;ENDFOLD
;FOLD LIN P193 CONT Vel=1 m/s CPDATP193 Tool[2] Base[10] ;%{PE}
;FOLD Parameters ;%{h}
;Params IlfProvider=kukaroboter.basistech.inlineforms.movement.old; Kuka.IsGlobalPoint=False; Kuka.PointName=P193; Kuka.BlendingEnabled=TRUE; Kuka.MoveDataName=CPDATP193; Kuka.VelocityPath=1; Kuka.CurrentCDSetIndex=0; Kuka.MovementParameterFieldEnabled=True; IlfCommand=LIN
;ENDFOLD
$BWDSTART = FALSE
LDAT_ACT=LCPDATP193
FDAT_ACT=FP193
BAS (#CP_PARAMS,1)
SET_CD_PARAMS (0)
LIN XP193 C_DIS

;ENDFOLD
;FOLD CIRC CAux194 CDes194 CONT Vel=0.1 m/s CPDATC194 Tool[2] Base[10] ;%{PE}
;FOLD Parameters ;%{h}
;Params IlfProvider=kukaroboter.basistech.inlineforms.movement.old; Kuka.IsGlobalPoint=False; Kuka.PointName=CDes194; Kuka.BlendingEnabled=TRUE; Kuka.MoveDataName=CPDATC194; Kuka.VelocityPath=0.1; Kuka.CurrentCDSetIndex=0; Kuka.MovementParameterFieldEnabled=True; IlfCommand=LIN
;ENDFOLD
$BWDSTART = FALSE
LDAT_ACT=LCPDATC194
FDAT_ACT=FC194
$ORI_TYPE = #VAR
$CIRC_TYPE = #PATH
BAS (#CP_PARAMS,0.1)
SET_CD_PARAMS (0)
CIRC XCAux194, XCDes194 C_DIS

;ENDFOLD
;FOLD LIN P195 CONT Vel=1 m/s CPDATP195 Tool[2] Base[10] ;%{PE}
;FOLD Parameters ;%{h}
;Params IlfProvider=kukaroboter.basistech.inlineforms.movement.old; Kuka.IsGlobalPoint=False; Kuka.PointName=P195; Kuka.BlendingEnabled=TRUE; Kuka.MoveDataName=CPDATP195; Kuka.VelocityPath=1; Kuka.CurrentCDSetIndex=0; Kuka.MovementParameterFieldEnabled=True; IlfCommand=LIN
;ENDFOLD
$BWDSTART = FALSE
LDAT_ACT=LCPDATP195
FDAT_ACT=FP195
BAS (#CP_PARAMS,1)
SET_CD_PARAMS (0)
LIN XP195 C_DIS

;ENDFOLD
;FOLD LIN P196 CONT Vel=1 m/s CPDATP196 Tool[2] Base[10] ;%{PE}
;FOLD Parameters ;%{h}
;Params IlfProvider=kukaroboter.basistech.inlineforms.movement.old; Kuka.IsGlobalPoint=False; Kuka.PointName=P196; Kuka.BlendingEnabled=TRUE; Kuka.MoveDataName=CPDATP196; Kuka.VelocityPath=1; Kuka.CurrentCDSetIndex=0; Kuka.MovementParameterFieldEnabled=True; IlfCommand=LIN
;ENDFOLD
$BWDSTART = FALSE
LDAT_ACT=LCPDATP196
FDAT_ACT=FP196
BAS (#CP_PARAMS,1)
SET_CD_PARAMS (0)
LIN XP196 C_DIS

;ENDFOLD
;FOLD CIRC CAux197 CDes197 CONT Vel=0.1 m/s CPDATC197 Tool[2] Base[10] ;%{PE}
;FOLD Parameters ;%{h}
;Params IlfProvider=kukaroboter.basistech.inlineforms.movement.old; Kuka.IsGlobalPoint=False; Kuka.PointName=CDes197; Kuka.BlendingEnabled=TRUE; Kuka.MoveDataName=CPDATC197; Kuka.VelocityPath=0.1; Kuka.CurrentCDSetIndex=0; Kuka.MovementParameterFieldEnabled=True; IlfCommand=LIN
;ENDFOLD
$BWDSTART = FALSE
LDAT_ACT=LCPDATC197
FDAT_ACT=FC197
$ORI_TYPE = #VAR
$CIRC_TYPE = #PATH
BAS (#CP_PARAMS,0.1)
SET_CD_PARAMS (0)
CIRC XCAux197, XCDes197 C_DIS

;ENDFOLD
;FOLD LIN P198 CONT Vel=1 m/s CPDATP198 Tool[2] Base[10] ;%{PE}
;FOLD Parameters ;%{h}
;Params IlfProvider=kukaroboter.basistech.inlineforms.movement.old; Kuka.IsGlobalPoint=False; Kuka.PointName=P198; Kuka.BlendingEnabled=TRUE; Kuka.MoveDataName=CPDATP198; Kuka.VelocityPath=1; Kuka.CurrentCDSetIndex=0; Kuka.MovementParameterFieldEnabled=True; IlfCommand=LIN
;ENDFOLD
$BWDSTART = FALSE
LDAT_ACT=LCPDATP198
FDAT_ACT=FP198
BAS (#CP_PARAMS,1)
SET_CD_PARAMS (0)
LIN XP198 C_DIS

;ENDFOLD
;FOLD LIN P199 CONT Vel=1 m/s CPDATP199 Tool[2] Base[10] ;%{PE}
;FOLD Parameters ;%{h}
;Params IlfProvider=kukaroboter.basistech.inlineforms.movement.old; Kuka.IsGlobalPoint=False; Kuka.PointName=P199; Kuka.BlendingEnabled=TRUE; Kuka.MoveDataName=CPDATP199; Kuka.VelocityPath=1; Kuka.CurrentCDSetIndex=0; Kuka.MovementParameterFieldEnabled=True; IlfCommand=LIN
;ENDFOLD
$BWDSTART = FALSE
LDAT_ACT=LCPDATP199
FDAT_ACT=FP199
BAS (#CP_PARAMS,1)
SET_CD_PARAMS (0)
LIN XP199 C_DIS

;ENDFOLD
;FOLD CIRC CAux200 CDes200 CONT Vel=0.1 m/s CPDATC200 Tool[2] Base[10] ;%{PE}
;FOLD Parameters ;%{h}
;Params IlfProvider=kukaroboter.basistech.inlineforms.movement.old; Kuka.IsGlobalPoint=False; Kuka.PointName=CDes200; Kuka.BlendingEnabled=TRUE; Kuka.MoveDataName=CPDATC200; Kuka.VelocityPath=0.1; Kuka.CurrentCDSetIndex=0; Kuka.MovementParameterFieldEnabled=True; IlfCommand=LIN
;ENDFOLD
$BWDSTART = FALSE
LDAT_ACT=LCPDATC200
FDAT_ACT=FC200
$ORI_TYPE = #VAR
$CIRC_TYPE = #PATH
BAS (#CP_PARAMS,0.1)
SET_CD_PARAMS (0)
CIRC XCAux200, XCDes200 C_DIS

;ENDFOLD
;FOLD LIN P201 CONT Vel=1 m/s CPDATP201 Tool[2] Base[10] ;%{PE}
;FOLD Parameters ;%{h}
;Params IlfProvider=kukaroboter.basistech.inlineforms.movement.old; Kuka.IsGlobalPoint=False; Kuka.PointName=P201; Kuka.BlendingEnabled=TRUE; Kuka.MoveDataName=CPDATP201; Kuka.VelocityPath=1; Kuka.CurrentCDSetIndex=0; Kuka.MovementParameterFieldEnabled=True; IlfCommand=LIN
;ENDFOLD
$BWDSTART = FALSE
LDAT_ACT=LCPDATP201
FDAT_ACT=FP201
BAS (#CP_PARAMS,1)
SET_CD_PARAMS (0)
LIN XP201 C_DIS

;ENDFOLD
;FOLD LIN P202 CONT Vel=1 m/s CPDATP202 Tool[2] Base[10] ;%{PE}
;FOLD Parameters ;%{h}
;Params IlfProvider=kukaroboter.basistech.inlineforms.movement.old; Kuka.IsGlobalPoint=False; Kuka.PointName=P202; Kuka.BlendingEnabled=TRUE; Kuka.MoveDataName=CPDATP202; Kuka.VelocityPath=1; Kuka.CurrentCDSetIndex=0; Kuka.MovementParameterFieldEnabled=True; IlfCommand=LIN
;ENDFOLD
$BWDSTART = FALSE
LDAT_ACT=LCPDATP202
FDAT_ACT=FP202
BAS (#CP_PARAMS,1)
SET_CD_PARAMS (0)
LIN XP202 C_DIS

;ENDFOLD
;FOLD CIRC CAux203 CDes203 CONT Vel=0.1 m/s CPDATC203 Tool[2] Base[10] ;%{PE}
;FOLD Parameters ;%{h}
;Params IlfProvider=kukaroboter.basistech.inlineforms.movement.old; Kuka.IsGlobalPoint=False; Kuka.PointName=CDes203; Kuka.BlendingEnabled=TRUE; Kuka.MoveDataName=CPDATC203; Kuka.VelocityPath=0.1; Kuka.CurrentCDSetIndex=0; Kuka.MovementParameterFieldEnabled=True; IlfCommand=LIN
;ENDFOLD
$BWDSTART = FALSE
LDAT_ACT=LCPDATC203
FDAT_ACT=FC203
$ORI_TYPE = #VAR
$CIRC_TYPE = #PATH
BAS (#CP_PARAMS,0.1)
SET_CD_PARAMS (0)
CIRC XCAux203, XCDes203 C_DIS

;ENDFOLD
;FOLD LIN P204 CONT Vel=1 m/s CPDATP204 Tool[2] Base[10] ;%{PE}
;FOLD Parameters ;%{h}
;Params IlfProvider=kukaroboter.basistech.inlineforms.movement.old; Kuka.IsGlobalPoint=False; Kuka.PointName=P204; Kuka.BlendingEnabled=TRUE; Kuka.MoveDataName=CPDATP204; Kuka.VelocityPath=1; Kuka.CurrentCDSetIndex=0; Kuka.MovementParameterFieldEnabled=True; IlfCommand=LIN
;ENDFOLD
$BWDSTART = FALSE
LDAT_ACT=LCPDATP204
FDAT_ACT=FP204
BAS (#CP_PARAMS,1)
SET_CD_PARAMS (0)
LIN XP204 C_DIS

;ENDFOLD
;FOLD LIN P205 CONT Vel=1 m/s CPDATP205 Tool[2] Base[10] ;%{PE}
;FOLD Parameters ;%{h}
;Params IlfProvider=kukaroboter.basistech.inlineforms.movement.old; Kuka.IsGlobalPoint=False; Kuka.PointName=P205; Kuka.BlendingEnabled=TRUE; Kuka.MoveDataName=CPDATP205; Kuka.VelocityPath=1; Kuka.CurrentCDSetIndex=0; Kuka.MovementParameterFieldEnabled=True; IlfCommand=LIN
;ENDFOLD
$BWDSTART = FALSE
LDAT_ACT=LCPDATP205
FDAT_ACT=FP205
BAS (#CP_PARAMS,1)
SET_CD_PARAMS (0)
LIN XP205 C_DIS

;ENDFOLD
;FOLD CIRC CAux206 CDes206 CONT Vel=0.1 m/s CPDATC206 Tool[2] Base[10] ;%{PE}
;FOLD Parameters ;%{h}
;Params IlfProvider=kukaroboter.basistech.inlineforms.movement.old; Kuka.IsGlobalPoint=False; Kuka.PointName=CDes206; Kuka.BlendingEnabled=TRUE; Kuka.MoveDataName=CPDATC206; Kuka.VelocityPath=0.1; Kuka.CurrentCDSetIndex=0; Kuka.MovementParameterFieldEnabled=True; IlfCommand=LIN
;ENDFOLD
$BWDSTART = FALSE
LDAT_ACT=LCPDATC206
FDAT_ACT=FC206
$ORI_TYPE = #VAR
$CIRC_TYPE = #PATH
BAS (#CP_PARAMS,0.1)
SET_CD_PARAMS (0)
CIRC XCAux206, XCDes206 C_DIS

;ENDFOLD
;FOLD LIN P207 CONT Vel=1 m/s CPDATP207 Tool[2] Base[10] ;%{PE}
;FOLD Parameters ;%{h}
;Params IlfProvider=kukaroboter.basistech.inlineforms.movement.old; Kuka.IsGlobalPoint=False; Kuka.PointName=P207; Kuka.BlendingEnabled=TRUE; Kuka.MoveDataName=CPDATP207; Kuka.VelocityPath=1; Kuka.CurrentCDSetIndex=0; Kuka.MovementParameterFieldEnabled=True; IlfCommand=LIN
;ENDFOLD
$BWDSTART = FALSE
LDAT_ACT=LCPDATP207
FDAT_ACT=FP207
BAS (#CP_PARAMS,1)
SET_CD_PARAMS (0)
LIN XP207 C_DIS

;ENDFOLD
;FOLD LIN P208 CONT Vel=1 m/s CPDATP208 Tool[2] Base[10] ;%{PE}
;FOLD Parameters ;%{h}
;Params IlfProvider=kukaroboter.basistech.inlineforms.movement.old; Kuka.IsGlobalPoint=False; Kuka.PointName=P208; Kuka.BlendingEnabled=TRUE; Kuka.MoveDataName=CPDATP208; Kuka.VelocityPath=1; Kuka.CurrentCDSetIndex=0; Kuka.MovementParameterFieldEnabled=True; IlfCommand=LIN
;ENDFOLD
$BWDSTART = FALSE
LDAT_ACT=LCPDATP208
FDAT_ACT=FP208
BAS (#CP_PARAMS,1)
SET_CD_PARAMS (0)
LIN XP208 C_DIS

;ENDFOLD
;FOLD CIRC CAux209 CDes209 CONT Vel=0.1 m/s CPDATC209 Tool[2] Base[10] ;%{PE}
;FOLD Parameters ;%{h}
;Params IlfProvider=kukaroboter.basistech.inlineforms.movement.old; Kuka.IsGlobalPoint=False; Kuka.PointName=CDes209; Kuka.BlendingEnabled=TRUE; Kuka.MoveDataName=CPDATC209; Kuka.VelocityPath=0.1; Kuka.CurrentCDSetIndex=0; Kuka.MovementParameterFieldEnabled=True; IlfCommand=LIN
;ENDFOLD
$BWDSTART = FALSE
LDAT_ACT=LCPDATC209
FDAT_ACT=FC209
$ORI_TYPE = #VAR
$CIRC_TYPE = #PATH
BAS (#CP_PARAMS,0.1)
SET_CD_PARAMS (0)
CIRC XCAux209, XCDes209 C_DIS

;ENDFOLD
;FOLD LIN P210 CONT Vel=1 m/s CPDATP210 Tool[2] Base[10] ;%{PE}
;FOLD Parameters ;%{h}
;Params IlfProvider=kukaroboter.basistech.inlineforms.movement.old; Kuka.IsGlobalPoint=False; Kuka.PointName=P210; Kuka.BlendingEnabled=TRUE; Kuka.MoveDataName=CPDATP210; Kuka.VelocityPath=1; Kuka.CurrentCDSetIndex=0; Kuka.MovementParameterFieldEnabled=True; IlfCommand=LIN
;ENDFOLD
$BWDSTART = FALSE
LDAT_ACT=LCPDATP210
FDAT_ACT=FP210
BAS (#CP_PARAMS,1)
SET_CD_PARAMS (0)
LIN XP210 C_DIS

;ENDFOLD
;FOLD LIN P211 CONT Vel=1 m/s CPDATP211 Tool[2] Base[10] ;%{PE}
;FOLD Parameters ;%{h}
;Params IlfProvider=kukaroboter.basistech.inlineforms.movement.old; Kuka.IsGlobalPoint=False; Kuka.PointName=P211; Kuka.BlendingEnabled=TRUE; Kuka.MoveDataName=CPDATP211; Kuka.VelocityPath=1; Kuka.CurrentCDSetIndex=0; Kuka.MovementParameterFieldEnabled=True; IlfCommand=LIN
;ENDFOLD
$BWDSTART = FALSE
LDAT_ACT=LCPDATP211
FDAT_ACT=FP211
BAS (#CP_PARAMS,1)
SET_CD_PARAMS (0)
LIN XP211 C_DIS

;ENDFOLD
;FOLD CIRC CAux212 CDes212 CONT Vel=0.1 m/s CPDATC212 Tool[2] Base[10] ;%{PE}
;FOLD Parameters ;%{h}
;Params IlfProvider=kukaroboter.basistech.inlineforms.movement.old; Kuka.IsGlobalPoint=False; Kuka.PointName=CDes212; Kuka.BlendingEnabled=TRUE; Kuka.MoveDataName=CPDATC212; Kuka.VelocityPath=0.1; Kuka.CurrentCDSetIndex=0; Kuka.MovementParameterFieldEnabled=True; IlfCommand=LIN
;ENDFOLD
$BWDSTART = FALSE
LDAT_ACT=LCPDATC212
FDAT_ACT=FC212
$ORI_TYPE = #VAR
$CIRC_TYPE = #PATH
BAS (#CP_PARAMS,0.1)
SET_CD_PARAMS (0)
CIRC XCAux212, XCDes212 C_DIS

;ENDFOLD
;FOLD LIN P213 CONT Vel=1 m/s CPDATP213 Tool[2] Base[10] ;%{PE}
;FOLD Parameters ;%{h}
;Params IlfProvider=kukaroboter.basistech.inlineforms.movement.old; Kuka.IsGlobalPoint=False; Kuka.PointName=P213; Kuka.BlendingEnabled=TRUE; Kuka.MoveDataName=CPDATP213; Kuka.VelocityPath=1; Kuka.CurrentCDSetIndex=0; Kuka.MovementParameterFieldEnabled=True; IlfCommand=LIN
;ENDFOLD
$BWDSTART = FALSE
LDAT_ACT=LCPDATP213
FDAT_ACT=FP213
BAS (#CP_PARAMS,1)
SET_CD_PARAMS (0)
LIN XP213 C_DIS

;ENDFOLD
;FOLD LIN P214 CONT Vel=1 m/s CPDATP214 Tool[2] Base[10] ;%{PE}
;FOLD Parameters ;%{h}
;Params IlfProvider=kukaroboter.basistech.inlineforms.movement.old; Kuka.IsGlobalPoint=False; Kuka.PointName=P214; Kuka.BlendingEnabled=TRUE; Kuka.MoveDataName=CPDATP214; Kuka.VelocityPath=1; Kuka.CurrentCDSetIndex=0; Kuka.MovementParameterFieldEnabled=True; IlfCommand=LIN
;ENDFOLD
$BWDSTART = FALSE
LDAT_ACT=LCPDATP214
FDAT_ACT=FP214
BAS (#CP_PARAMS,1)
SET_CD_PARAMS (0)
LIN XP214 C_DIS

;ENDFOLD
;FOLD CIRC CAux215 CDes215 CONT Vel=0.1 m/s CPDATC215 Tool[2] Base[10] ;%{PE}
;FOLD Parameters ;%{h}
;Params IlfProvider=kukaroboter.basistech.inlineforms.movement.old; Kuka.IsGlobalPoint=False; Kuka.PointName=CDes215; Kuka.BlendingEnabled=TRUE; Kuka.MoveDataName=CPDATC215; Kuka.VelocityPath=0.1; Kuka.CurrentCDSetIndex=0; Kuka.MovementParameterFieldEnabled=True; IlfCommand=LIN
;ENDFOLD
$BWDSTART = FALSE
LDAT_ACT=LCPDATC215
FDAT_ACT=FC215
$ORI_TYPE = #VAR
$CIRC_TYPE = #PATH
BAS (#CP_PARAMS,0.1)
SET_CD_PARAMS (0)
CIRC XCAux215, XCDes215 C_DIS

;ENDFOLD
;FOLD LIN P216 CONT Vel=1 m/s CPDATP216 Tool[2] Base[10] ;%{PE}
;FOLD Parameters ;%{h}
;Params IlfProvider=kukaroboter.basistech.inlineforms.movement.old; Kuka.IsGlobalPoint=False; Kuka.PointName=P216; Kuka.BlendingEnabled=TRUE; Kuka.MoveDataName=CPDATP216; Kuka.VelocityPath=1; Kuka.CurrentCDSetIndex=0; Kuka.MovementParameterFieldEnabled=True; IlfCommand=LIN
;ENDFOLD
$BWDSTART = FALSE
LDAT_ACT=LCPDATP216
FDAT_ACT=FP216
BAS (#CP_PARAMS,1)
SET_CD_PARAMS (0)
LIN XP216 C_DIS

;ENDFOLD
;FOLD LIN P217 CONT Vel=1 m/s CPDATP217 Tool[2] Base[10] ;%{PE}
;FOLD Parameters ;%{h}
;Params IlfProvider=kukaroboter.basistech.inlineforms.movement.old; Kuka.IsGlobalPoint=False; Kuka.PointName=P217; Kuka.BlendingEnabled=TRUE; Kuka.MoveDataName=CPDATP217; Kuka.VelocityPath=1; Kuka.CurrentCDSetIndex=0; Kuka.MovementParameterFieldEnabled=True; IlfCommand=LIN
;ENDFOLD
$BWDSTART = FALSE
LDAT_ACT=LCPDATP217
FDAT_ACT=FP217
BAS (#CP_PARAMS,1)
SET_CD_PARAMS (0)
LIN XP217 C_DIS

;ENDFOLD
;FOLD CIRC CAux218 CDes218 CONT Vel=0.1 m/s CPDATC218 Tool[2] Base[10] ;%{PE}
;FOLD Parameters ;%{h}
;Params IlfProvider=kukaroboter.basistech.inlineforms.movement.old; Kuka.IsGlobalPoint=False; Kuka.PointName=CDes218; Kuka.BlendingEnabled=TRUE; Kuka.MoveDataName=CPDATC218; Kuka.VelocityPath=0.1; Kuka.CurrentCDSetIndex=0; Kuka.MovementParameterFieldEnabled=True; IlfCommand=LIN
;ENDFOLD
$BWDSTART = FALSE
LDAT_ACT=LCPDATC218
FDAT_ACT=FC218
$ORI_TYPE = #VAR
$CIRC_TYPE = #PATH
BAS (#CP_PARAMS,0.1)
SET_CD_PARAMS (0)
CIRC XCAux218, XCDes218 C_DIS

;ENDFOLD
;FOLD LIN P219 CONT Vel=1 m/s CPDATP219 Tool[2] Base[10] ;%{PE}
;FOLD Parameters ;%{h}
;Params IlfProvider=kukaroboter.basistech.inlineforms.movement.old; Kuka.IsGlobalPoint=False; Kuka.PointName=P219; Kuka.BlendingEnabled=TRUE; Kuka.MoveDataName=CPDATP219; Kuka.VelocityPath=1; Kuka.CurrentCDSetIndex=0; Kuka.MovementParameterFieldEnabled=True; IlfCommand=LIN
;ENDFOLD
$BWDSTART = FALSE
LDAT_ACT=LCPDATP219
FDAT_ACT=FP219
BAS (#CP_PARAMS,1)
SET_CD_PARAMS (0)
LIN XP219 C_DIS

;ENDFOLD
;FOLD LIN P220 CONT Vel=1 m/s CPDATP220 Tool[2] Base[10] ;%{PE}
;FOLD Parameters ;%{h}
;Params IlfProvider=kukaroboter.basistech.inlineforms.movement.old; Kuka.IsGlobalPoint=False; Kuka.PointName=P220; Kuka.BlendingEnabled=TRUE; Kuka.MoveDataName=CPDATP220; Kuka.VelocityPath=1; Kuka.CurrentCDSetIndex=0; Kuka.MovementParameterFieldEnabled=True; IlfCommand=LIN
;ENDFOLD
$BWDSTART = FALSE
LDAT_ACT=LCPDATP220
FDAT_ACT=FP220
BAS (#CP_PARAMS,1)
SET_CD_PARAMS (0)
LIN XP220 C_DIS

;ENDFOLD
;FOLD CIRC CAux221 CDes221 CONT Vel=0.1 m/s CPDATC221 Tool[2] Base[10] ;%{PE}
;FOLD Parameters ;%{h}
;Params IlfProvider=kukaroboter.basistech.inlineforms.movement.old; Kuka.IsGlobalPoint=False; Kuka.PointName=CDes221; Kuka.BlendingEnabled=TRUE; Kuka.MoveDataName=CPDATC221; Kuka.VelocityPath=0.1; Kuka.CurrentCDSetIndex=0; Kuka.MovementParameterFieldEnabled=True; IlfCommand=LIN
;ENDFOLD
$BWDSTART = FALSE
LDAT_ACT=LCPDATC221
FDAT_ACT=FC221
$ORI_TYPE = #VAR
$CIRC_TYPE = #PATH
BAS (#CP_PARAMS,0.1)
SET_CD_PARAMS (0)
CIRC XCAux221, XCDes221 C_DIS

;ENDFOLD
;FOLD LIN P222 CONT Vel=1 m/s CPDATP222 Tool[2] Base[10] ;%{PE}
;FOLD Parameters ;%{h}
;Params IlfProvider=kukaroboter.basistech.inlineforms.movement.old; Kuka.IsGlobalPoint=False; Kuka.PointName=P222; Kuka.BlendingEnabled=TRUE; Kuka.MoveDataName=CPDATP222; Kuka.VelocityPath=1; Kuka.CurrentCDSetIndex=0; Kuka.MovementParameterFieldEnabled=True; IlfCommand=LIN
;ENDFOLD
$BWDSTART = FALSE
LDAT_ACT=LCPDATP222
FDAT_ACT=FP222
BAS (#CP_PARAMS,1)
SET_CD_PARAMS (0)
LIN XP222 C_DIS

;ENDFOLD
;FOLD LIN P223 CONT Vel=1 m/s CPDATP223 Tool[2] Base[10] ;%{PE}
;FOLD Parameters ;%{h}
;Params IlfProvider=kukaroboter.basistech.inlineforms.movement.old; Kuka.IsGlobalPoint=False; Kuka.PointName=P223; Kuka.BlendingEnabled=TRUE; Kuka.MoveDataName=CPDATP223; Kuka.VelocityPath=1; Kuka.CurrentCDSetIndex=0; Kuka.MovementParameterFieldEnabled=True; IlfCommand=LIN
;ENDFOLD
$BWDSTART = FALSE
LDAT_ACT=LCPDATP223
FDAT_ACT=FP223
BAS (#CP_PARAMS,1)
SET_CD_PARAMS (0)
LIN XP223 C_DIS

;ENDFOLD
;FOLD CIRC CAux224 CDes224 CONT Vel=0.1 m/s CPDATC224 Tool[2] Base[10] ;%{PE}
;FOLD Parameters ;%{h}
;Params IlfProvider=kukaroboter.basistech.inlineforms.movement.old; Kuka.IsGlobalPoint=False; Kuka.PointName=CDes224; Kuka.BlendingEnabled=TRUE; Kuka.MoveDataName=CPDATC224; Kuka.VelocityPath=0.1; Kuka.CurrentCDSetIndex=0; Kuka.MovementParameterFieldEnabled=True; IlfCommand=LIN
;ENDFOLD
$BWDSTART = FALSE
LDAT_ACT=LCPDATC224
FDAT_ACT=FC224
$ORI_TYPE = #VAR
$CIRC_TYPE = #PATH
BAS (#CP_PARAMS,0.1)
SET_CD_PARAMS (0)
CIRC XCAux224, XCDes224 C_DIS

;ENDFOLD
;FOLD LIN P225 CONT Vel=1 m/s CPDATP225 Tool[2] Base[10] ;%{PE}
;FOLD Parameters ;%{h}
;Params IlfProvider=kukaroboter.basistech.inlineforms.movement.old; Kuka.IsGlobalPoint=False; Kuka.PointName=P225; Kuka.BlendingEnabled=TRUE; Kuka.MoveDataName=CPDATP225; Kuka.VelocityPath=1; Kuka.CurrentCDSetIndex=0; Kuka.MovementParameterFieldEnabled=True; IlfCommand=LIN
;ENDFOLD
$BWDSTART = FALSE
LDAT_ACT=LCPDATP225
FDAT_ACT=FP225
BAS (#CP_PARAMS,1)
SET_CD_PARAMS (0)
LIN XP225 C_DIS

;ENDFOLD
;FOLD LIN P226 CONT Vel=1 m/s CPDATP226 Tool[2] Base[10] ;%{PE}
;FOLD Parameters ;%{h}
;Params IlfProvider=kukaroboter.basistech.inlineforms.movement.old; Kuka.IsGlobalPoint=False; Kuka.PointName=P226; Kuka.BlendingEnabled=TRUE; Kuka.MoveDataName=CPDATP226; Kuka.VelocityPath=1; Kuka.CurrentCDSetIndex=0; Kuka.MovementParameterFieldEnabled=True; IlfCommand=LIN
;ENDFOLD
$BWDSTART = FALSE
LDAT_ACT=LCPDATP226
FDAT_ACT=FP226
BAS (#CP_PARAMS,1)
SET_CD_PARAMS (0)
LIN XP226 C_DIS

;ENDFOLD
;FOLD CIRC CAux227 CDes227 CONT Vel=0.1 m/s CPDATC227 Tool[2] Base[10] ;%{PE}
;FOLD Parameters ;%{h}
;Params IlfProvider=kukaroboter.basistech.inlineforms.movement.old; Kuka.IsGlobalPoint=False; Kuka.PointName=CDes227; Kuka.BlendingEnabled=TRUE; Kuka.MoveDataName=CPDATC227; Kuka.VelocityPath=0.1; Kuka.CurrentCDSetIndex=0; Kuka.MovementParameterFieldEnabled=True; IlfCommand=LIN
;ENDFOLD
$BWDSTART = FALSE
LDAT_ACT=LCPDATC227
FDAT_ACT=FC227
$ORI_TYPE = #VAR
$CIRC_TYPE = #PATH
BAS (#CP_PARAMS,0.1)
SET_CD_PARAMS (0)
CIRC XCAux227, XCDes227 C_DIS

;ENDFOLD
;FOLD LIN P228 CONT Vel=1 m/s CPDATP228 Tool[2] Base[10] ;%{PE}
;FOLD Parameters ;%{h}
;Params IlfProvider=kukaroboter.basistech.inlineforms.movement.old; Kuka.IsGlobalPoint=False; Kuka.PointName=P228; Kuka.BlendingEnabled=TRUE; Kuka.MoveDataName=CPDATP228; Kuka.VelocityPath=1; Kuka.CurrentCDSetIndex=0; Kuka.MovementParameterFieldEnabled=True; IlfCommand=LIN
;ENDFOLD
$BWDSTART = FALSE
LDAT_ACT=LCPDATP228
FDAT_ACT=FP228
BAS (#CP_PARAMS,1)
SET_CD_PARAMS (0)
LIN XP228 C_DIS

;ENDFOLD
;FOLD LIN P229 CONT Vel=1 m/s CPDATP229 Tool[2] Base[10] ;%{PE}
;FOLD Parameters ;%{h}
;Params IlfProvider=kukaroboter.basistech.inlineforms.movement.old; Kuka.IsGlobalPoint=False; Kuka.PointName=P229; Kuka.BlendingEnabled=TRUE; Kuka.MoveDataName=CPDATP229; Kuka.VelocityPath=1; Kuka.CurrentCDSetIndex=0; Kuka.MovementParameterFieldEnabled=True; IlfCommand=LIN
;ENDFOLD
$BWDSTART = FALSE
LDAT_ACT=LCPDATP229
FDAT_ACT=FP229
BAS (#CP_PARAMS,1)
SET_CD_PARAMS (0)
LIN XP229 C_DIS

;ENDFOLD
;FOLD CIRC CAux230 CDes230 CONT Vel=0.1 m/s CPDATC230 Tool[2] Base[10] ;%{PE}
;FOLD Parameters ;%{h}
;Params IlfProvider=kukaroboter.basistech.inlineforms.movement.old; Kuka.IsGlobalPoint=False; Kuka.PointName=CDes230; Kuka.BlendingEnabled=TRUE; Kuka.MoveDataName=CPDATC230; Kuka.VelocityPath=0.1; Kuka.CurrentCDSetIndex=0; Kuka.MovementParameterFieldEnabled=True; IlfCommand=LIN
;ENDFOLD
$BWDSTART = FALSE
LDAT_ACT=LCPDATC230
FDAT_ACT=FC230
$ORI_TYPE = #VAR
$CIRC_TYPE = #PATH
BAS (#CP_PARAMS,0.1)
SET_CD_PARAMS (0)
CIRC XCAux230, XCDes230 C_DIS

;ENDFOLD
;FOLD LIN P231 CONT Vel=1 m/s CPDATP231 Tool[2] Base[10] ;%{PE}
;FOLD Parameters ;%{h}
;Params IlfProvider=kukaroboter.basistech.inlineforms.movement.old; Kuka.IsGlobalPoint=False; Kuka.PointName=P231; Kuka.BlendingEnabled=TRUE; Kuka.MoveDataName=CPDATP231; Kuka.VelocityPath=1; Kuka.CurrentCDSetIndex=0; Kuka.MovementParameterFieldEnabled=True; IlfCommand=LIN
;ENDFOLD
$BWDSTART = FALSE
LDAT_ACT=LCPDATP231
FDAT_ACT=FP231
BAS (#CP_PARAMS,1)
SET_CD_PARAMS (0)
LIN XP231 C_DIS

;ENDFOLD
;FOLD LIN P232 CONT Vel=1 m/s CPDATP232 Tool[2] Base[10] ;%{PE}
;FOLD Parameters ;%{h}
;Params IlfProvider=kukaroboter.basistech.inlineforms.movement.old; Kuka.IsGlobalPoint=False; Kuka.PointName=P232; Kuka.BlendingEnabled=TRUE; Kuka.MoveDataName=CPDATP232; Kuka.VelocityPath=1; Kuka.CurrentCDSetIndex=0; Kuka.MovementParameterFieldEnabled=True; IlfCommand=LIN
;ENDFOLD
$BWDSTART = FALSE
LDAT_ACT=LCPDATP232
FDAT_ACT=FP232
BAS (#CP_PARAMS,1)
SET_CD_PARAMS (0)
LIN XP232 C_DIS

;ENDFOLD
;FOLD CIRC CAux233 CDes233 CONT Vel=0.1 m/s CPDATC233 Tool[2] Base[10] ;%{PE}
;FOLD Parameters ;%{h}
;Params IlfProvider=kukaroboter.basistech.inlineforms.movement.old; Kuka.IsGlobalPoint=False; Kuka.PointName=CDes233; Kuka.BlendingEnabled=TRUE; Kuka.MoveDataName=CPDATC233; Kuka.VelocityPath=0.1; Kuka.CurrentCDSetIndex=0; Kuka.MovementParameterFieldEnabled=True; IlfCommand=LIN
;ENDFOLD
$BWDSTART = FALSE
LDAT_ACT=LCPDATC233
FDAT_ACT=FC233
$ORI_TYPE = #VAR
$CIRC_TYPE = #PATH
BAS (#CP_PARAMS,0.1)
SET_CD_PARAMS (0)
CIRC XCAux233, XCDes233 C_DIS

;ENDFOLD
;FOLD LIN P234 CONT Vel=1 m/s CPDATP234 Tool[2] Base[10] ;%{PE}
;FOLD Parameters ;%{h}
;Params IlfProvider=kukaroboter.basistech.inlineforms.movement.old; Kuka.IsGlobalPoint=False; Kuka.PointName=P234; Kuka.BlendingEnabled=TRUE; Kuka.MoveDataName=CPDATP234; Kuka.VelocityPath=1; Kuka.CurrentCDSetIndex=0; Kuka.MovementParameterFieldEnabled=True; IlfCommand=LIN
;ENDFOLD
$BWDSTART = FALSE
LDAT_ACT=LCPDATP234
FDAT_ACT=FP234
BAS (#CP_PARAMS,1)
SET_CD_PARAMS (0)
LIN XP234 C_DIS

;ENDFOLD
;FOLD LIN P235 CONT Vel=1 m/s CPDATP235 Tool[2] Base[10] ;%{PE}
;FOLD Parameters ;%{h}
;Params IlfProvider=kukaroboter.basistech.inlineforms.movement.old; Kuka.IsGlobalPoint=False; Kuka.PointName=P235; Kuka.BlendingEnabled=TRUE; Kuka.MoveDataName=CPDATP235; Kuka.VelocityPath=1; Kuka.CurrentCDSetIndex=0; Kuka.MovementParameterFieldEnabled=True; IlfCommand=LIN
;ENDFOLD
$BWDSTART = FALSE
LDAT_ACT=LCPDATP235
FDAT_ACT=FP235
BAS (#CP_PARAMS,1)
SET_CD_PARAMS (0)
LIN XP235 C_DIS

;ENDFOLD
;FOLD CIRC CAux236 CDes236 CONT Vel=0.1 m/s CPDATC236 Tool[2] Base[10] ;%{PE}
;FOLD Parameters ;%{h}
;Params IlfProvider=kukaroboter.basistech.inlineforms.movement.old; Kuka.IsGlobalPoint=False; Kuka.PointName=CDes236; Kuka.BlendingEnabled=TRUE; Kuka.MoveDataName=CPDATC236; Kuka.VelocityPath=0.1; Kuka.CurrentCDSetIndex=0; Kuka.MovementParameterFieldEnabled=True; IlfCommand=LIN
;ENDFOLD
$BWDSTART = FALSE
LDAT_ACT=LCPDATC236
FDAT_ACT=FC236
$ORI_TYPE = #VAR
$CIRC_TYPE = #PATH
BAS (#CP_PARAMS,0.1)
SET_CD_PARAMS (0)
CIRC XCAux236, XCDes236 C_DIS

;ENDFOLD
;FOLD LIN P237 CONT Vel=1 m/s CPDATP237 Tool[2] Base[10] ;%{PE}
;FOLD Parameters ;%{h}
;Params IlfProvider=kukaroboter.basistech.inlineforms.movement.old; Kuka.IsGlobalPoint=False; Kuka.PointName=P237; Kuka.BlendingEnabled=TRUE; Kuka.MoveDataName=CPDATP237; Kuka.VelocityPath=1; Kuka.CurrentCDSetIndex=0; Kuka.MovementParameterFieldEnabled=True; IlfCommand=LIN
;ENDFOLD
$BWDSTART = FALSE
LDAT_ACT=LCPDATP237
FDAT_ACT=FP237
BAS (#CP_PARAMS,1)
SET_CD_PARAMS (0)
LIN XP237 C_DIS

;ENDFOLD
;FOLD LIN P238 CONT Vel=1 m/s CPDATP238 Tool[2] Base[10] ;%{PE}
;FOLD Parameters ;%{h}
;Params IlfProvider=kukaroboter.basistech.inlineforms.movement.old; Kuka.IsGlobalPoint=False; Kuka.PointName=P238; Kuka.BlendingEnabled=TRUE; Kuka.MoveDataName=CPDATP238; Kuka.VelocityPath=1; Kuka.CurrentCDSetIndex=0; Kuka.MovementParameterFieldEnabled=True; IlfCommand=LIN
;ENDFOLD
$BWDSTART = FALSE
LDAT_ACT=LCPDATP238
FDAT_ACT=FP238
BAS (#CP_PARAMS,1)
SET_CD_PARAMS (0)
LIN XP238 C_DIS

;ENDFOLD
;FOLD CIRC CAux239 CDes239 CONT Vel=0.1 m/s CPDATC239 Tool[2] Base[10] ;%{PE}
;FOLD Parameters ;%{h}
;Params IlfProvider=kukaroboter.basistech.inlineforms.movement.old; Kuka.IsGlobalPoint=False; Kuka.PointName=CDes239; Kuka.BlendingEnabled=TRUE; Kuka.MoveDataName=CPDATC239; Kuka.VelocityPath=0.1; Kuka.CurrentCDSetIndex=0; Kuka.MovementParameterFieldEnabled=True; IlfCommand=LIN
;ENDFOLD
$BWDSTART = FALSE
LDAT_ACT=LCPDATC239
FDAT_ACT=FC239
$ORI_TYPE = #VAR
$CIRC_TYPE = #PATH
BAS (#CP_PARAMS,0.1)
SET_CD_PARAMS (0)
CIRC XCAux239, XCDes239 C_DIS

;ENDFOLD
;FOLD LIN P240 CONT Vel=1 m/s CPDATP240 Tool[2] Base[10] ;%{PE}
;FOLD Parameters ;%{h}
;Params IlfProvider=kukaroboter.basistech.inlineforms.movement.old; Kuka.IsGlobalPoint=False; Kuka.PointName=P240; Kuka.BlendingEnabled=TRUE; Kuka.MoveDataName=CPDATP240; Kuka.VelocityPath=1; Kuka.CurrentCDSetIndex=0; Kuka.MovementParameterFieldEnabled=True; IlfCommand=LIN
;ENDFOLD
$BWDSTART = FALSE
LDAT_ACT=LCPDATP240
FDAT_ACT=FP240
BAS (#CP_PARAMS,1)
SET_CD_PARAMS (0)
LIN XP240 C_DIS

;ENDFOLD
;FOLD LIN P241 CONT Vel=1 m/s CPDATP241 Tool[2] Base[10] ;%{PE}
;FOLD Parameters ;%{h}
;Params IlfProvider=kukaroboter.basistech.inlineforms.movement.old; Kuka.IsGlobalPoint=False; Kuka.PointName=P241; Kuka.BlendingEnabled=TRUE; Kuka.MoveDataName=CPDATP241; Kuka.VelocityPath=1; Kuka.CurrentCDSetIndex=0; Kuka.MovementParameterFieldEnabled=True; IlfCommand=LIN
;ENDFOLD
$BWDSTART = FALSE
LDAT_ACT=LCPDATP241
FDAT_ACT=FP241
BAS (#CP_PARAMS,1)
SET_CD_PARAMS (0)
LIN XP241 C_DIS

;ENDFOLD
;FOLD CIRC CAux242 CDes242 CONT Vel=0.1 m/s CPDATC242 Tool[2] Base[10] ;%{PE}
;FOLD Parameters ;%{h}
;Params IlfProvider=kukaroboter.basistech.inlineforms.movement.old; Kuka.IsGlobalPoint=False; Kuka.PointName=CDes242; Kuka.BlendingEnabled=TRUE; Kuka.MoveDataName=CPDATC242; Kuka.VelocityPath=0.1; Kuka.CurrentCDSetIndex=0; Kuka.MovementParameterFieldEnabled=True; IlfCommand=LIN
;ENDFOLD
$BWDSTART = FALSE
LDAT_ACT=LCPDATC242
FDAT_ACT=FC242
$ORI_TYPE = #VAR
$CIRC_TYPE = #PATH
BAS (#CP_PARAMS,0.1)
SET_CD_PARAMS (0)
CIRC XCAux242, XCDes242 C_DIS

;ENDFOLD
;FOLD LIN P243 CONT Vel=1 m/s CPDATP243 Tool[2] Base[10] ;%{PE}
;FOLD Parameters ;%{h}
;Params IlfProvider=kukaroboter.basistech.inlineforms.movement.old; Kuka.IsGlobalPoint=False; Kuka.PointName=P243; Kuka.BlendingEnabled=TRUE; Kuka.MoveDataName=CPDATP243; Kuka.VelocityPath=1; Kuka.CurrentCDSetIndex=0; Kuka.MovementParameterFieldEnabled=True; IlfCommand=LIN
;ENDFOLD
$BWDSTART = FALSE
LDAT_ACT=LCPDATP243
FDAT_ACT=FP243
BAS (#CP_PARAMS,1)
SET_CD_PARAMS (0)
LIN XP243 C_DIS

;ENDFOLD
;FOLD LIN P244 CONT Vel=1 m/s CPDATP244 Tool[2] Base[10] ;%{PE}
;FOLD Parameters ;%{h}
;Params IlfProvider=kukaroboter.basistech.inlineforms.movement.old; Kuka.IsGlobalPoint=False; Kuka.PointName=P244; Kuka.BlendingEnabled=TRUE; Kuka.MoveDataName=CPDATP244; Kuka.VelocityPath=1; Kuka.CurrentCDSetIndex=0; Kuka.MovementParameterFieldEnabled=True; IlfCommand=LIN
;ENDFOLD
$BWDSTART = FALSE
LDAT_ACT=LCPDATP244
FDAT_ACT=FP244
BAS (#CP_PARAMS,1)
SET_CD_PARAMS (0)
LIN XP244 C_DIS

;ENDFOLD
;FOLD CIRC CAux245 CDes245 CONT Vel=0.1 m/s CPDATC245 Tool[2] Base[10] ;%{PE}
;FOLD Parameters ;%{h}
;Params IlfProvider=kukaroboter.basistech.inlineforms.movement.old; Kuka.IsGlobalPoint=False; Kuka.PointName=CDes245; Kuka.BlendingEnabled=TRUE; Kuka.MoveDataName=CPDATC245; Kuka.VelocityPath=0.1; Kuka.CurrentCDSetIndex=0; Kuka.MovementParameterFieldEnabled=True; IlfCommand=LIN
;ENDFOLD
$BWDSTART = FALSE
LDAT_ACT=LCPDATC245
FDAT_ACT=FC245
$ORI_TYPE = #VAR
$CIRC_TYPE = #PATH
BAS (#CP_PARAMS,0.1)
SET_CD_PARAMS (0)
CIRC XCAux245, XCDes245 C_DIS

;ENDFOLD
;FOLD LIN P246 CONT Vel=1 m/s CPDATP246 Tool[2] Base[10] ;%{PE}
;FOLD Parameters ;%{h}
;Params IlfProvider=kukaroboter.basistech.inlineforms.movement.old; Kuka.IsGlobalPoint=False; Kuka.PointName=P246; Kuka.BlendingEnabled=TRUE; Kuka.MoveDataName=CPDATP246; Kuka.VelocityPath=1; Kuka.CurrentCDSetIndex=0; Kuka.MovementParameterFieldEnabled=True; IlfCommand=LIN
;ENDFOLD
$BWDSTART = FALSE
LDAT_ACT=LCPDATP246
FDAT_ACT=FP246
BAS (#CP_PARAMS,1)
SET_CD_PARAMS (0)
LIN XP246 C_DIS

;ENDFOLD
;FOLD LIN P247 CONT Vel=1 m/s CPDATP247 Tool[2] Base[10] ;%{PE}
;FOLD Parameters ;%{h}
;Params IlfProvider=kukaroboter.basistech.inlineforms.movement.old; Kuka.IsGlobalPoint=False; Kuka.PointName=P247; Kuka.BlendingEnabled=TRUE; Kuka.MoveDataName=CPDATP247; Kuka.VelocityPath=1; Kuka.CurrentCDSetIndex=0; Kuka.MovementParameterFieldEnabled=True; IlfCommand=LIN
;ENDFOLD
$BWDSTART = FALSE
LDAT_ACT=LCPDATP247
FDAT_ACT=FP247
BAS (#CP_PARAMS,1)
SET_CD_PARAMS (0)
LIN XP247 C_DIS

;ENDFOLD
;FOLD CIRC CAux248 CDes248 CONT Vel=0.1 m/s CPDATC248 Tool[2] Base[10] ;%{PE}
;FOLD Parameters ;%{h}
;Params IlfProvider=kukaroboter.basistech.inlineforms.movement.old; Kuka.IsGlobalPoint=False; Kuka.PointName=CDes248; Kuka.BlendingEnabled=TRUE; Kuka.MoveDataName=CPDATC248; Kuka.VelocityPath=0.1; Kuka.CurrentCDSetIndex=0; Kuka.MovementParameterFieldEnabled=True; IlfCommand=LIN
;ENDFOLD
$BWDSTART = FALSE
LDAT_ACT=LCPDATC248
FDAT_ACT=FC248
$ORI_TYPE = #VAR
$CIRC_TYPE = #PATH
BAS (#CP_PARAMS,0.1)
SET_CD_PARAMS (0)
CIRC XCAux248, XCDes248 C_DIS

;ENDFOLD
;FOLD LIN P249 CONT Vel=1 m/s CPDATP249 Tool[2] Base[10] ;%{PE}
;FOLD Parameters ;%{h}
;Params IlfProvider=kukaroboter.basistech.inlineforms.movement.old; Kuka.IsGlobalPoint=False; Kuka.PointName=P249; Kuka.BlendingEnabled=TRUE; Kuka.MoveDataName=CPDATP249; Kuka.VelocityPath=1; Kuka.CurrentCDSetIndex=0; Kuka.MovementParameterFieldEnabled=True; IlfCommand=LIN
;ENDFOLD
$BWDSTART = FALSE
LDAT_ACT=LCPDATP249
FDAT_ACT=FP249
BAS (#CP_PARAMS,1)
SET_CD_PARAMS (0)
LIN XP249 C_DIS

;ENDFOLD
;FOLD LIN P250 CONT Vel=1 m/s CPDATP250 Tool[2] Base[10] ;%{PE}
;FOLD Parameters ;%{h}
;Params IlfProvider=kukaroboter.basistech.inlineforms.movement.old; Kuka.IsGlobalPoint=False; Kuka.PointName=P250; Kuka.BlendingEnabled=TRUE; Kuka.MoveDataName=CPDATP250; Kuka.VelocityPath=1; Kuka.CurrentCDSetIndex=0; Kuka.MovementParameterFieldEnabled=True; IlfCommand=LIN
;ENDFOLD
$BWDSTART = FALSE
LDAT_ACT=LCPDATP250
FDAT_ACT=FP250
BAS (#CP_PARAMS,1)
SET_CD_PARAMS (0)
LIN XP250 C_DIS

;ENDFOLD
;FOLD CIRC CAux251 CDes251 CONT Vel=0.1 m/s CPDATC251 Tool[2] Base[10] ;%{PE}
;FOLD Parameters ;%{h}
;Params IlfProvider=kukaroboter.basistech.inlineforms.movement.old; Kuka.IsGlobalPoint=False; Kuka.PointName=CDes251; Kuka.BlendingEnabled=TRUE; Kuka.MoveDataName=CPDATC251; Kuka.VelocityPath=0.1; Kuka.CurrentCDSetIndex=0; Kuka.MovementParameterFieldEnabled=True; IlfCommand=LIN
;ENDFOLD
$BWDSTART = FALSE
LDAT_ACT=LCPDATC251
FDAT_ACT=FC251
$ORI_TYPE = #VAR
$CIRC_TYPE = #PATH
BAS (#CP_PARAMS,0.1)
SET_CD_PARAMS (0)
CIRC XCAux251, XCDes251 C_DIS

;ENDFOLD
;FOLD LIN P252 CONT Vel=1 m/s CPDATP252 Tool[2] Base[10] ;%{PE}
;FOLD Parameters ;%{h}
;Params IlfProvider=kukaroboter.basistech.inlineforms.movement.old; Kuka.IsGlobalPoint=False; Kuka.PointName=P252; Kuka.BlendingEnabled=TRUE; Kuka.MoveDataName=CPDATP252; Kuka.VelocityPath=1; Kuka.CurrentCDSetIndex=0; Kuka.MovementParameterFieldEnabled=True; IlfCommand=LIN
;ENDFOLD
$BWDSTART = FALSE
LDAT_ACT=LCPDATP252
FDAT_ACT=FP252
BAS (#CP_PARAMS,1)
SET_CD_PARAMS (0)
LIN XP252 C_DIS

;ENDFOLD
;FOLD LIN P253 CONT Vel=1 m/s CPDATP253 Tool[2] Base[10] ;%{PE}
;FOLD Parameters ;%{h}
;Params IlfProvider=kukaroboter.basistech.inlineforms.movement.old; Kuka.IsGlobalPoint=False; Kuka.PointName=P253; Kuka.BlendingEnabled=TRUE; Kuka.MoveDataName=CPDATP253; Kuka.VelocityPath=1; Kuka.CurrentCDSetIndex=0; Kuka.MovementParameterFieldEnabled=True; IlfCommand=LIN
;ENDFOLD
$BWDSTART = FALSE
LDAT_ACT=LCPDATP253
FDAT_ACT=FP253
BAS (#CP_PARAMS,1)
SET_CD_PARAMS (0)
LIN XP253 C_DIS

;ENDFOLD
;FOLD CIRC CAux254 CDes254 CONT Vel=0.1 m/s CPDATC254 Tool[2] Base[10] ;%{PE}
;FOLD Parameters ;%{h}
;Params IlfProvider=kukaroboter.basistech.inlineforms.movement.old; Kuka.IsGlobalPoint=False; Kuka.PointName=CDes254; Kuka.BlendingEnabled=TRUE; Kuka.MoveDataName=CPDATC254; Kuka.VelocityPath=0.1; Kuka.CurrentCDSetIndex=0; Kuka.MovementParameterFieldEnabled=True; IlfCommand=LIN
;ENDFOLD
$BWDSTART = FALSE
LDAT_ACT=LCPDATC254
FDAT_ACT=FC254
$ORI_TYPE = #VAR
$CIRC_TYPE = #PATH
BAS (#CP_PARAMS,0.1)
SET_CD_PARAMS (0)
CIRC XCAux254, XCDes254 C_DIS

;ENDFOLD
;FOLD LIN P255 CONT Vel=1 m/s CPDATP255 Tool[2] Base[10] ;%{PE}
;FOLD Parameters ;%{h}
;Params IlfProvider=kukaroboter.basistech.inlineforms.movement.old; Kuka.IsGlobalPoint=False; Kuka.PointName=P255; Kuka.BlendingEnabled=TRUE; Kuka.MoveDataName=CPDATP255; Kuka.VelocityPath=1; Kuka.CurrentCDSetIndex=0; Kuka.MovementParameterFieldEnabled=True; IlfCommand=LIN
;ENDFOLD
$BWDSTART = FALSE
LDAT_ACT=LCPDATP255
FDAT_ACT=FP255
BAS (#CP_PARAMS,1)
SET_CD_PARAMS (0)
LIN XP255 C_DIS

;ENDFOLD
;FOLD LIN P256 CONT Vel=1 m/s CPDATP256 Tool[2] Base[10] ;%{PE}
;FOLD Parameters ;%{h}
;Params IlfProvider=kukaroboter.basistech.inlineforms.movement.old; Kuka.IsGlobalPoint=False; Kuka.PointName=P256; Kuka.BlendingEnabled=TRUE; Kuka.MoveDataName=CPDATP256; Kuka.VelocityPath=1; Kuka.CurrentCDSetIndex=0; Kuka.MovementParameterFieldEnabled=True; IlfCommand=LIN
;ENDFOLD
$BWDSTART = FALSE
LDAT_ACT=LCPDATP256
FDAT_ACT=FP256
BAS (#CP_PARAMS,1)
SET_CD_PARAMS (0)
LIN XP256 C_DIS

;ENDFOLD
;FOLD CIRC CAux257 CDes257 CONT Vel=0.1 m/s CPDATC257 Tool[2] Base[10] ;%{PE}
;FOLD Parameters ;%{h}
;Params IlfProvider=kukaroboter.basistech.inlineforms.movement.old; Kuka.IsGlobalPoint=False; Kuka.PointName=CDes257; Kuka.BlendingEnabled=TRUE; Kuka.MoveDataName=CPDATC257; Kuka.VelocityPath=0.1; Kuka.CurrentCDSetIndex=0; Kuka.MovementParameterFieldEnabled=True; IlfCommand=LIN
;ENDFOLD
$BWDSTART = FALSE
LDAT_ACT=LCPDATC257
FDAT_ACT=FC257
$ORI_TYPE = #VAR
$CIRC_TYPE = #PATH
BAS (#CP_PARAMS,0.1)
SET_CD_PARAMS (0)
CIRC XCAux257, XCDes257 C_DIS

;ENDFOLD
;FOLD LIN P258 CONT Vel=1 m/s CPDATP258 Tool[2] Base[10] ;%{PE}
;FOLD Parameters ;%{h}
;Params IlfProvider=kukaroboter.basistech.inlineforms.movement.old; Kuka.IsGlobalPoint=False; Kuka.PointName=P258; Kuka.BlendingEnabled=TRUE; Kuka.MoveDataName=CPDATP258; Kuka.VelocityPath=1; Kuka.CurrentCDSetIndex=0; Kuka.MovementParameterFieldEnabled=True; IlfCommand=LIN
;ENDFOLD
$BWDSTART = FALSE
LDAT_ACT=LCPDATP258
FDAT_ACT=FP258
BAS (#CP_PARAMS,1)
SET_CD_PARAMS (0)
LIN XP258 C_DIS

;ENDFOLD
;FOLD LIN P259 CONT Vel=1 m/s CPDATP259 Tool[2] Base[10] ;%{PE}
;FOLD Parameters ;%{h}
;Params IlfProvider=kukaroboter.basistech.inlineforms.movement.old; Kuka.IsGlobalPoint=False; Kuka.PointName=P259; Kuka.BlendingEnabled=TRUE; Kuka.MoveDataName=CPDATP259; Kuka.VelocityPath=1; Kuka.CurrentCDSetIndex=0; Kuka.MovementParameterFieldEnabled=True; IlfCommand=LIN
;ENDFOLD
$BWDSTART = FALSE
LDAT_ACT=LCPDATP259
FDAT_ACT=FP259
BAS (#CP_PARAMS,1)
SET_CD_PARAMS (0)
LIN XP259 C_DIS

;ENDFOLD
;FOLD CIRC CAux260 CDes260 CONT Vel=0.1 m/s CPDATC260 Tool[2] Base[10] ;%{PE}
;FOLD Parameters ;%{h}
;Params IlfProvider=kukaroboter.basistech.inlineforms.movement.old; Kuka.IsGlobalPoint=False; Kuka.PointName=CDes260; Kuka.BlendingEnabled=TRUE; Kuka.MoveDataName=CPDATC260; Kuka.VelocityPath=0.1; Kuka.CurrentCDSetIndex=0; Kuka.MovementParameterFieldEnabled=True; IlfCommand=LIN
;ENDFOLD
$BWDSTART = FALSE
LDAT_ACT=LCPDATC260
FDAT_ACT=FC260
$ORI_TYPE = #VAR
$CIRC_TYPE = #PATH
BAS (#CP_PARAMS,0.1)
SET_CD_PARAMS (0)
CIRC XCAux260, XCDes260 C_DIS

;ENDFOLD
;FOLD LIN P261 CONT Vel=1 m/s CPDATP261 Tool[2] Base[10] ;%{PE}
;FOLD Parameters ;%{h}
;Params IlfProvider=kukaroboter.basistech.inlineforms.movement.old; Kuka.IsGlobalPoint=False; Kuka.PointName=P261; Kuka.BlendingEnabled=TRUE; Kuka.MoveDataName=CPDATP261; Kuka.VelocityPath=1; Kuka.CurrentCDSetIndex=0; Kuka.MovementParameterFieldEnabled=True; IlfCommand=LIN
;ENDFOLD
$BWDSTART = FALSE
LDAT_ACT=LCPDATP261
FDAT_ACT=FP261
BAS (#CP_PARAMS,1)
SET_CD_PARAMS (0)
LIN XP261 C_DIS

;ENDFOLD
;FOLD LIN P262 CONT Vel=1 m/s CPDATP262 Tool[2] Base[10] ;%{PE}
;FOLD Parameters ;%{h}
;Params IlfProvider=kukaroboter.basistech.inlineforms.movement.old; Kuka.IsGlobalPoint=False; Kuka.PointName=P262; Kuka.BlendingEnabled=TRUE; Kuka.MoveDataName=CPDATP262; Kuka.VelocityPath=1; Kuka.CurrentCDSetIndex=0; Kuka.MovementParameterFieldEnabled=True; IlfCommand=LIN
;ENDFOLD
$BWDSTART = FALSE
LDAT_ACT=LCPDATP262
FDAT_ACT=FP262
BAS (#CP_PARAMS,1)
SET_CD_PARAMS (0)
LIN XP262 C_DIS

;ENDFOLD
;FOLD CIRC CAux263 CDes263 CONT Vel=0.1 m/s CPDATC263 Tool[2] Base[10] ;%{PE}
;FOLD Parameters ;%{h}
;Params IlfProvider=kukaroboter.basistech.inlineforms.movement.old; Kuka.IsGlobalPoint=False; Kuka.PointName=CDes263; Kuka.BlendingEnabled=TRUE; Kuka.MoveDataName=CPDATC263; Kuka.VelocityPath=0.1; Kuka.CurrentCDSetIndex=0; Kuka.MovementParameterFieldEnabled=True; IlfCommand=LIN
;ENDFOLD
$BWDSTART = FALSE
LDAT_ACT=LCPDATC263
FDAT_ACT=FC263
$ORI_TYPE = #VAR
$CIRC_TYPE = #PATH
BAS (#CP_PARAMS,0.1)
SET_CD_PARAMS (0)
CIRC XCAux263, XCDes263 C_DIS

;ENDFOLD
;FOLD LIN P264 CONT Vel=1 m/s CPDATP264 Tool[2] Base[10] ;%{PE}
;FOLD Parameters ;%{h}
;Params IlfProvider=kukaroboter.basistech.inlineforms.movement.old; Kuka.IsGlobalPoint=False; Kuka.PointName=P264; Kuka.BlendingEnabled=TRUE; Kuka.MoveDataName=CPDATP264; Kuka.VelocityPath=1; Kuka.CurrentCDSetIndex=0; Kuka.MovementParameterFieldEnabled=True; IlfCommand=LIN
;ENDFOLD
$BWDSTART = FALSE
LDAT_ACT=LCPDATP264
FDAT_ACT=FP264
BAS (#CP_PARAMS,1)
SET_CD_PARAMS (0)
LIN XP264 C_DIS

;ENDFOLD
;FOLD LIN P265 CONT Vel=1 m/s CPDATP265 Tool[2] Base[10] ;%{PE}
;FOLD Parameters ;%{h}
;Params IlfProvider=kukaroboter.basistech.inlineforms.movement.old; Kuka.IsGlobalPoint=False; Kuka.PointName=P265; Kuka.BlendingEnabled=TRUE; Kuka.MoveDataName=CPDATP265; Kuka.VelocityPath=1; Kuka.CurrentCDSetIndex=0; Kuka.MovementParameterFieldEnabled=True; IlfCommand=LIN
;ENDFOLD
$BWDSTART = FALSE
LDAT_ACT=LCPDATP265
FDAT_ACT=FP265
BAS (#CP_PARAMS,1)
SET_CD_PARAMS (0)
LIN XP265 C_DIS

;ENDFOLD
;FOLD CIRC CAux266 CDes266 CONT Vel=0.1 m/s CPDATC266 Tool[2] Base[10] ;%{PE}
;FOLD Parameters ;%{h}
;Params IlfProvider=kukaroboter.basistech.inlineforms.movement.old; Kuka.IsGlobalPoint=False; Kuka.PointName=CDes266; Kuka.BlendingEnabled=TRUE; Kuka.MoveDataName=CPDATC266; Kuka.VelocityPath=0.1; Kuka.CurrentCDSetIndex=0; Kuka.MovementParameterFieldEnabled=True; IlfCommand=LIN
;ENDFOLD
$BWDSTART = FALSE
LDAT_ACT=LCPDATC266
FDAT_ACT=FC266
$ORI_TYPE = #VAR
$CIRC_TYPE = #PATH
BAS (#CP_PARAMS,0.1)
SET_CD_PARAMS (0)
CIRC XCAux266, XCDes266 C_DIS

;ENDFOLD
;FOLD LIN P267 CONT Vel=1 m/s CPDATP267 Tool[2] Base[10] ;%{PE}
;FOLD Parameters ;%{h}
;Params IlfProvider=kukaroboter.basistech.inlineforms.movement.old; Kuka.IsGlobalPoint=False; Kuka.PointName=P267; Kuka.BlendingEnabled=TRUE; Kuka.MoveDataName=CPDATP267; Kuka.VelocityPath=1; Kuka.CurrentCDSetIndex=0; Kuka.MovementParameterFieldEnabled=True; IlfCommand=LIN
;ENDFOLD
$BWDSTART = FALSE
LDAT_ACT=LCPDATP267
FDAT_ACT=FP267
BAS (#CP_PARAMS,1)
SET_CD_PARAMS (0)
LIN XP267 C_DIS

;ENDFOLD
;FOLD LIN P268 CONT Vel=1 m/s CPDATP268 Tool[2] Base[10] ;%{PE}
;FOLD Parameters ;%{h}
;Params IlfProvider=kukaroboter.basistech.inlineforms.movement.old; Kuka.IsGlobalPoint=False; Kuka.PointName=P268; Kuka.BlendingEnabled=TRUE; Kuka.MoveDataName=CPDATP268; Kuka.VelocityPath=1; Kuka.CurrentCDSetIndex=0; Kuka.MovementParameterFieldEnabled=True; IlfCommand=LIN
;ENDFOLD
$BWDSTART = FALSE
LDAT_ACT=LCPDATP268
FDAT_ACT=FP268
BAS (#CP_PARAMS,1)
SET_CD_PARAMS (0)
LIN XP268 C_DIS

;ENDFOLD
;FOLD CIRC CAux269 CDes269 CONT Vel=0.1 m/s CPDATC269 Tool[2] Base[10] ;%{PE}
;FOLD Parameters ;%{h}
;Params IlfProvider=kukaroboter.basistech.inlineforms.movement.old; Kuka.IsGlobalPoint=False; Kuka.PointName=CDes269; Kuka.BlendingEnabled=TRUE; Kuka.MoveDataName=CPDATC269; Kuka.VelocityPath=0.1; Kuka.CurrentCDSetIndex=0; Kuka.MovementParameterFieldEnabled=True; IlfCommand=LIN
;ENDFOLD
$BWDSTART = FALSE
LDAT_ACT=LCPDATC269
FDAT_ACT=FC269
$ORI_TYPE = #VAR
$CIRC_TYPE = #PATH
BAS (#CP_PARAMS,0.1)
SET_CD_PARAMS (0)
CIRC XCAux269, XCDes269 C_DIS

;ENDFOLD
;FOLD LIN P270 CONT Vel=1 m/s CPDATP270 Tool[2] Base[10] ;%{PE}
;FOLD Parameters ;%{h}
;Params IlfProvider=kukaroboter.basistech.inlineforms.movement.old; Kuka.IsGlobalPoint=False; Kuka.PointName=P270; Kuka.BlendingEnabled=TRUE; Kuka.MoveDataName=CPDATP270; Kuka.VelocityPath=1; Kuka.CurrentCDSetIndex=0; Kuka.MovementParameterFieldEnabled=True; IlfCommand=LIN
;ENDFOLD
$BWDSTART = FALSE
LDAT_ACT=LCPDATP270
FDAT_ACT=FP270
BAS (#CP_PARAMS,1)
SET_CD_PARAMS (0)
LIN XP270 C_DIS

;ENDFOLD
;FOLD LIN P271 CONT Vel=1 m/s CPDATP271 Tool[2] Base[10] ;%{PE}
;FOLD Parameters ;%{h}
;Params IlfProvider=kukaroboter.basistech.inlineforms.movement.old; Kuka.IsGlobalPoint=False; Kuka.PointName=P271; Kuka.BlendingEnabled=TRUE; Kuka.MoveDataName=CPDATP271; Kuka.VelocityPath=1; Kuka.CurrentCDSetIndex=0; Kuka.MovementParameterFieldEnabled=True; IlfCommand=LIN
;ENDFOLD
$BWDSTART = FALSE
LDAT_ACT=LCPDATP271
FDAT_ACT=FP271
BAS (#CP_PARAMS,1)
SET_CD_PARAMS (0)
LIN XP271 C_DIS

;ENDFOLD
;FOLD CIRC CAux272 CDes272 CONT Vel=0.1 m/s CPDATC272 Tool[2] Base[10] ;%{PE}
;FOLD Parameters ;%{h}
;Params IlfProvider=kukaroboter.basistech.inlineforms.movement.old; Kuka.IsGlobalPoint=False; Kuka.PointName=CDes272; Kuka.BlendingEnabled=TRUE; Kuka.MoveDataName=CPDATC272; Kuka.VelocityPath=0.1; Kuka.CurrentCDSetIndex=0; Kuka.MovementParameterFieldEnabled=True; IlfCommand=LIN
;ENDFOLD
$BWDSTART = FALSE
LDAT_ACT=LCPDATC272
FDAT_ACT=FC272
$ORI_TYPE = #VAR
$CIRC_TYPE = #PATH
BAS (#CP_PARAMS,0.1)
SET_CD_PARAMS (0)
CIRC XCAux272, XCDes272 C_DIS

;ENDFOLD
;FOLD LIN P273 CONT Vel=1 m/s CPDATP273 Tool[2] Base[10] ;%{PE}
;FOLD Parameters ;%{h}
;Params IlfProvider=kukaroboter.basistech.inlineforms.movement.old; Kuka.IsGlobalPoint=False; Kuka.PointName=P273; Kuka.BlendingEnabled=TRUE; Kuka.MoveDataName=CPDATP273; Kuka.VelocityPath=1; Kuka.CurrentCDSetIndex=0; Kuka.MovementParameterFieldEnabled=True; IlfCommand=LIN
;ENDFOLD
$BWDSTART = FALSE
LDAT_ACT=LCPDATP273
FDAT_ACT=FP273
BAS (#CP_PARAMS,1)
SET_CD_PARAMS (0)
LIN XP273 C_DIS

;ENDFOLD
;FOLD LIN P274 CONT Vel=1 m/s CPDATP274 Tool[2] Base[10] ;%{PE}
;FOLD Parameters ;%{h}
;Params IlfProvider=kukaroboter.basistech.inlineforms.movement.old; Kuka.IsGlobalPoint=False; Kuka.PointName=P274; Kuka.BlendingEnabled=TRUE; Kuka.MoveDataName=CPDATP274; Kuka.VelocityPath=1; Kuka.CurrentCDSetIndex=0; Kuka.MovementParameterFieldEnabled=True; IlfCommand=LIN
;ENDFOLD
$BWDSTART = FALSE
LDAT_ACT=LCPDATP274
FDAT_ACT=FP274
BAS (#CP_PARAMS,1)
SET_CD_PARAMS (0)
LIN XP274 C_DIS

;ENDFOLD
;FOLD CIRC CAux275 CDes275 CONT Vel=0.1 m/s CPDATC275 Tool[2] Base[10] ;%{PE}
;FOLD Parameters ;%{h}
;Params IlfProvider=kukaroboter.basistech.inlineforms.movement.old; Kuka.IsGlobalPoint=False; Kuka.PointName=CDes275; Kuka.BlendingEnabled=TRUE; Kuka.MoveDataName=CPDATC275; Kuka.VelocityPath=0.1; Kuka.CurrentCDSetIndex=0; Kuka.MovementParameterFieldEnabled=True; IlfCommand=LIN
;ENDFOLD
$BWDSTART = FALSE
LDAT_ACT=LCPDATC275
FDAT_ACT=FC275
$ORI_TYPE = #VAR
$CIRC_TYPE = #PATH
BAS (#CP_PARAMS,0.1)
SET_CD_PARAMS (0)
CIRC XCAux275, XCDes275 C_DIS

;ENDFOLD
;FOLD LIN P276 CONT Vel=1 m/s CPDATP276 Tool[2] Base[10] ;%{PE}
;FOLD Parameters ;%{h}
;Params IlfProvider=kukaroboter.basistech.inlineforms.movement.old; Kuka.IsGlobalPoint=False; Kuka.PointName=P276; Kuka.BlendingEnabled=TRUE; Kuka.MoveDataName=CPDATP276; Kuka.VelocityPath=1; Kuka.CurrentCDSetIndex=0; Kuka.MovementParameterFieldEnabled=True; IlfCommand=LIN
;ENDFOLD
$BWDSTART = FALSE
LDAT_ACT=LCPDATP276
FDAT_ACT=FP276
BAS (#CP_PARAMS,1)
SET_CD_PARAMS (0)
LIN XP276 C_DIS

;ENDFOLD
;FOLD LIN P277 CONT Vel=1 m/s CPDATP277 Tool[2] Base[10] ;%{PE}
;FOLD Parameters ;%{h}
;Params IlfProvider=kukaroboter.basistech.inlineforms.movement.old; Kuka.IsGlobalPoint=False; Kuka.PointName=P277; Kuka.BlendingEnabled=TRUE; Kuka.MoveDataName=CPDATP277; Kuka.VelocityPath=1; Kuka.CurrentCDSetIndex=0; Kuka.MovementParameterFieldEnabled=True; IlfCommand=LIN
;ENDFOLD
$BWDSTART = FALSE
LDAT_ACT=LCPDATP277
FDAT_ACT=FP277
BAS (#CP_PARAMS,1)
SET_CD_PARAMS (0)
LIN XP277 C_DIS

;ENDFOLD
;FOLD CIRC CAux278 CDes278 CONT Vel=0.1 m/s CPDATC278 Tool[2] Base[10] ;%{PE}
;FOLD Parameters ;%{h}
;Params IlfProvider=kukaroboter.basistech.inlineforms.movement.old; Kuka.IsGlobalPoint=False; Kuka.PointName=CDes278; Kuka.BlendingEnabled=TRUE; Kuka.MoveDataName=CPDATC278; Kuka.VelocityPath=0.1; Kuka.CurrentCDSetIndex=0; Kuka.MovementParameterFieldEnabled=True; IlfCommand=LIN
;ENDFOLD
$BWDSTART = FALSE
LDAT_ACT=LCPDATC278
FDAT_ACT=FC278
$ORI_TYPE = #VAR
$CIRC_TYPE = #PATH
BAS (#CP_PARAMS,0.1)
SET_CD_PARAMS (0)
CIRC XCAux278, XCDes278 C_DIS

;ENDFOLD
;FOLD LIN P279 CONT Vel=1 m/s CPDATP279 Tool[2] Base[10] ;%{PE}
;FOLD Parameters ;%{h}
;Params IlfProvider=kukaroboter.basistech.inlineforms.movement.old; Kuka.IsGlobalPoint=False; Kuka.PointName=P279; Kuka.BlendingEnabled=TRUE; Kuka.MoveDataName=CPDATP279; Kuka.VelocityPath=1; Kuka.CurrentCDSetIndex=0; Kuka.MovementParameterFieldEnabled=True; IlfCommand=LIN
;ENDFOLD
$BWDSTART = FALSE
LDAT_ACT=LCPDATP279
FDAT_ACT=FP279
BAS (#CP_PARAMS,1)
SET_CD_PARAMS (0)
LIN XP279 C_DIS

;ENDFOLD
;FOLD LIN P280 CONT Vel=1 m/s CPDATP280 Tool[2] Base[10] ;%{PE}
;FOLD Parameters ;%{h}
;Params IlfProvider=kukaroboter.basistech.inlineforms.movement.old; Kuka.IsGlobalPoint=False; Kuka.PointName=P280; Kuka.BlendingEnabled=TRUE; Kuka.MoveDataName=CPDATP280; Kuka.VelocityPath=1; Kuka.CurrentCDSetIndex=0; Kuka.MovementParameterFieldEnabled=True; IlfCommand=LIN
;ENDFOLD
$BWDSTART = FALSE
LDAT_ACT=LCPDATP280
FDAT_ACT=FP280
BAS (#CP_PARAMS,1)
SET_CD_PARAMS (0)
LIN XP280 C_DIS

;ENDFOLD
;FOLD CIRC CAux281 CDes281 CONT Vel=0.1 m/s CPDATC281 Tool[2] Base[10] ;%{PE}
;FOLD Parameters ;%{h}
;Params IlfProvider=kukaroboter.basistech.inlineforms.movement.old; Kuka.IsGlobalPoint=False; Kuka.PointName=CDes281; Kuka.BlendingEnabled=TRUE; Kuka.MoveDataName=CPDATC281; Kuka.VelocityPath=0.1; Kuka.CurrentCDSetIndex=0; Kuka.MovementParameterFieldEnabled=True; IlfCommand=LIN
;ENDFOLD
$BWDSTART = FALSE
LDAT_ACT=LCPDATC281
FDAT_ACT=FC281
$ORI_TYPE = #VAR
$CIRC_TYPE = #PATH
BAS (#CP_PARAMS,0.1)
SET_CD_PARAMS (0)
CIRC XCAux281, XCDes281 C_DIS

;ENDFOLD
;FOLD LIN P282 CONT Vel=1 m/s CPDATP282 Tool[2] Base[10] ;%{PE}
;FOLD Parameters ;%{h}
;Params IlfProvider=kukaroboter.basistech.inlineforms.movement.old; Kuka.IsGlobalPoint=False; Kuka.PointName=P282; Kuka.BlendingEnabled=TRUE; Kuka.MoveDataName=CPDATP282; Kuka.VelocityPath=1; Kuka.CurrentCDSetIndex=0; Kuka.MovementParameterFieldEnabled=True; IlfCommand=LIN
;ENDFOLD
$BWDSTART = FALSE
LDAT_ACT=LCPDATP282
FDAT_ACT=FP282
BAS (#CP_PARAMS,1)
SET_CD_PARAMS (0)
LIN XP282 C_DIS

;ENDFOLD
;FOLD LIN P283 CONT Vel=1 m/s CPDATP283 Tool[2] Base[10] ;%{PE}
;FOLD Parameters ;%{h}
;Params IlfProvider=kukaroboter.basistech.inlineforms.movement.old; Kuka.IsGlobalPoint=False; Kuka.PointName=P283; Kuka.BlendingEnabled=TRUE; Kuka.MoveDataName=CPDATP283; Kuka.VelocityPath=1; Kuka.CurrentCDSetIndex=0; Kuka.MovementParameterFieldEnabled=True; IlfCommand=LIN
;ENDFOLD
$BWDSTART = FALSE
LDAT_ACT=LCPDATP283
FDAT_ACT=FP283
BAS (#CP_PARAMS,1)
SET_CD_PARAMS (0)
LIN XP283 C_DIS

;ENDFOLD
;FOLD CIRC CAux284 CDes284 CONT Vel=0.1 m/s CPDATC284 Tool[2] Base[10] ;%{PE}
;FOLD Parameters ;%{h}
;Params IlfProvider=kukaroboter.basistech.inlineforms.movement.old; Kuka.IsGlobalPoint=False; Kuka.PointName=CDes284; Kuka.BlendingEnabled=TRUE; Kuka.MoveDataName=CPDATC284; Kuka.VelocityPath=0.1; Kuka.CurrentCDSetIndex=0; Kuka.MovementParameterFieldEnabled=True; IlfCommand=LIN
;ENDFOLD
$BWDSTART = FALSE
LDAT_ACT=LCPDATC284
FDAT_ACT=FC284
$ORI_TYPE = #VAR
$CIRC_TYPE = #PATH
BAS (#CP_PARAMS,0.1)
SET_CD_PARAMS (0)
CIRC XCAux284, XCDes284 C_DIS

;ENDFOLD
;FOLD LIN P285 CONT Vel=1 m/s CPDATP285 Tool[2] Base[10] ;%{PE}
;FOLD Parameters ;%{h}
;Params IlfProvider=kukaroboter.basistech.inlineforms.movement.old; Kuka.IsGlobalPoint=False; Kuka.PointName=P285; Kuka.BlendingEnabled=TRUE; Kuka.MoveDataName=CPDATP285; Kuka.VelocityPath=1; Kuka.CurrentCDSetIndex=0; Kuka.MovementParameterFieldEnabled=True; IlfCommand=LIN
;ENDFOLD
$BWDSTART = FALSE
LDAT_ACT=LCPDATP285
FDAT_ACT=FP285
BAS (#CP_PARAMS,1)
SET_CD_PARAMS (0)
LIN XP285 C_DIS

;ENDFOLD
;FOLD LIN P286 CONT Vel=1 m/s CPDATP286 Tool[2] Base[10] ;%{PE}
;FOLD Parameters ;%{h}
;Params IlfProvider=kukaroboter.basistech.inlineforms.movement.old; Kuka.IsGlobalPoint=False; Kuka.PointName=P286; Kuka.BlendingEnabled=TRUE; Kuka.MoveDataName=CPDATP286; Kuka.VelocityPath=1; Kuka.CurrentCDSetIndex=0; Kuka.MovementParameterFieldEnabled=True; IlfCommand=LIN
;ENDFOLD
$BWDSTART = FALSE
LDAT_ACT=LCPDATP286
FDAT_ACT=FP286
BAS (#CP_PARAMS,1)
SET_CD_PARAMS (0)
LIN XP286 C_DIS

;ENDFOLD
;FOLD CIRC CAux287 CDes287 CONT Vel=0.1 m/s CPDATC287 Tool[2] Base[10] ;%{PE}
;FOLD Parameters ;%{h}
;Params IlfProvider=kukaroboter.basistech.inlineforms.movement.old; Kuka.IsGlobalPoint=False; Kuka.PointName=CDes287; Kuka.BlendingEnabled=TRUE; Kuka.MoveDataName=CPDATC287; Kuka.VelocityPath=0.1; Kuka.CurrentCDSetIndex=0; Kuka.MovementParameterFieldEnabled=True; IlfCommand=LIN
;ENDFOLD
$BWDSTART = FALSE
LDAT_ACT=LCPDATC287
FDAT_ACT=FC287
$ORI_TYPE = #VAR
$CIRC_TYPE = #PATH
BAS (#CP_PARAMS,0.1)
SET_CD_PARAMS (0)
CIRC XCAux287, XCDes287 C_DIS

;ENDFOLD
;FOLD LIN P288 CONT Vel=1 m/s CPDATP288 Tool[2] Base[10] ;%{PE}
;FOLD Parameters ;%{h}
;Params IlfProvider=kukaroboter.basistech.inlineforms.movement.old; Kuka.IsGlobalPoint=False; Kuka.PointName=P288; Kuka.BlendingEnabled=TRUE; Kuka.MoveDataName=CPDATP288; Kuka.VelocityPath=1; Kuka.CurrentCDSetIndex=0; Kuka.MovementParameterFieldEnabled=True; IlfCommand=LIN
;ENDFOLD
$BWDSTART = FALSE
LDAT_ACT=LCPDATP288
FDAT_ACT=FP288
BAS (#CP_PARAMS,1)
SET_CD_PARAMS (0)
LIN XP288 C_DIS

;ENDFOLD
;FOLD LIN P289 CONT Vel=1 m/s CPDATP289 Tool[2] Base[10] ;%{PE}
;FOLD Parameters ;%{h}
;Params IlfProvider=kukaroboter.basistech.inlineforms.movement.old; Kuka.IsGlobalPoint=False; Kuka.PointName=P289; Kuka.BlendingEnabled=TRUE; Kuka.MoveDataName=CPDATP289; Kuka.VelocityPath=1; Kuka.CurrentCDSetIndex=0; Kuka.MovementParameterFieldEnabled=True; IlfCommand=LIN
;ENDFOLD
$BWDSTART = FALSE
LDAT_ACT=LCPDATP289
FDAT_ACT=FP289
BAS (#CP_PARAMS,1)
SET_CD_PARAMS (0)
LIN XP289 C_DIS

;ENDFOLD
;FOLD CIRC CAux290 CDes290 CONT Vel=0.1 m/s CPDATC290 Tool[2] Base[10] ;%{PE}
;FOLD Parameters ;%{h}
;Params IlfProvider=kukaroboter.basistech.inlineforms.movement.old; Kuka.IsGlobalPoint=False; Kuka.PointName=CDes290; Kuka.BlendingEnabled=TRUE; Kuka.MoveDataName=CPDATC290; Kuka.VelocityPath=0.1; Kuka.CurrentCDSetIndex=0; Kuka.MovementParameterFieldEnabled=True; IlfCommand=LIN
;ENDFOLD
$BWDSTART = FALSE
LDAT_ACT=LCPDATC290
FDAT_ACT=FC290
$ORI_TYPE = #VAR
$CIRC_TYPE = #PATH
BAS (#CP_PARAMS,0.1)
SET_CD_PARAMS (0)
CIRC XCAux290, XCDes290 C_DIS

;ENDFOLD
;FOLD LIN P291 CONT Vel=1 m/s CPDATP291 Tool[2] Base[10] ;%{PE}
;FOLD Parameters ;%{h}
;Params IlfProvider=kukaroboter.basistech.inlineforms.movement.old; Kuka.IsGlobalPoint=False; Kuka.PointName=P291; Kuka.BlendingEnabled=TRUE; Kuka.MoveDataName=CPDATP291; Kuka.VelocityPath=1; Kuka.CurrentCDSetIndex=0; Kuka.MovementParameterFieldEnabled=True; IlfCommand=LIN
;ENDFOLD
$BWDSTART = FALSE
LDAT_ACT=LCPDATP291
FDAT_ACT=FP291
BAS (#CP_PARAMS,1)
SET_CD_PARAMS (0)
LIN XP291 C_DIS

;ENDFOLD
;FOLD LIN P292 CONT Vel=1 m/s CPDATP292 Tool[2] Base[10] ;%{PE}
;FOLD Parameters ;%{h}
;Params IlfProvider=kukaroboter.basistech.inlineforms.movement.old; Kuka.IsGlobalPoint=False; Kuka.PointName=P292; Kuka.BlendingEnabled=TRUE; Kuka.MoveDataName=CPDATP292; Kuka.VelocityPath=1; Kuka.CurrentCDSetIndex=0; Kuka.MovementParameterFieldEnabled=True; IlfCommand=LIN
;ENDFOLD
$BWDSTART = FALSE
LDAT_ACT=LCPDATP292
FDAT_ACT=FP292
BAS (#CP_PARAMS,1)
SET_CD_PARAMS (0)
LIN XP292 C_DIS

;ENDFOLD
;FOLD CIRC CAux293 CDes293 CONT Vel=0.1 m/s CPDATC293 Tool[2] Base[10] ;%{PE}
;FOLD Parameters ;%{h}
;Params IlfProvider=kukaroboter.basistech.inlineforms.movement.old; Kuka.IsGlobalPoint=False; Kuka.PointName=CDes293; Kuka.BlendingEnabled=TRUE; Kuka.MoveDataName=CPDATC293; Kuka.VelocityPath=0.1; Kuka.CurrentCDSetIndex=0; Kuka.MovementParameterFieldEnabled=True; IlfCommand=LIN
;ENDFOLD
$BWDSTART = FALSE
LDAT_ACT=LCPDATC293
FDAT_ACT=FC293
$ORI_TYPE = #VAR
$CIRC_TYPE = #PATH
BAS (#CP_PARAMS,0.1)
SET_CD_PARAMS (0)
CIRC XCAux293, XCDes293 C_DIS

;ENDFOLD
;FOLD LIN P294 CONT Vel=1 m/s CPDATP294 Tool[2] Base[10] ;%{PE}
;FOLD Parameters ;%{h}
;Params IlfProvider=kukaroboter.basistech.inlineforms.movement.old; Kuka.IsGlobalPoint=False; Kuka.PointName=P294; Kuka.BlendingEnabled=TRUE; Kuka.MoveDataName=CPDATP294; Kuka.VelocityPath=1; Kuka.CurrentCDSetIndex=0; Kuka.MovementParameterFieldEnabled=True; IlfCommand=LIN
;ENDFOLD
$BWDSTART = FALSE
LDAT_ACT=LCPDATP294
FDAT_ACT=FP294
BAS (#CP_PARAMS,1)
SET_CD_PARAMS (0)
LIN XP294 C_DIS

;ENDFOLD
;FOLD LIN P295 CONT Vel=1 m/s CPDATP295 Tool[2] Base[10] ;%{PE}
;FOLD Parameters ;%{h}
;Params IlfProvider=kukaroboter.basistech.inlineforms.movement.old; Kuka.IsGlobalPoint=False; Kuka.PointName=P295; Kuka.BlendingEnabled=TRUE; Kuka.MoveDataName=CPDATP295; Kuka.VelocityPath=1; Kuka.CurrentCDSetIndex=0; Kuka.MovementParameterFieldEnabled=True; IlfCommand=LIN
;ENDFOLD
$BWDSTART = FALSE
LDAT_ACT=LCPDATP295
FDAT_ACT=FP295
BAS (#CP_PARAMS,1)
SET_CD_PARAMS (0)
LIN XP295 C_DIS

;ENDFOLD
;FOLD CIRC CAux296 CDes296 CONT Vel=0.1 m/s CPDATC296 Tool[2] Base[10] ;%{PE}
;FOLD Parameters ;%{h}
;Params IlfProvider=kukaroboter.basistech.inlineforms.movement.old; Kuka.IsGlobalPoint=False; Kuka.PointName=CDes296; Kuka.BlendingEnabled=TRUE; Kuka.MoveDataName=CPDATC296; Kuka.VelocityPath=0.1; Kuka.CurrentCDSetIndex=0; Kuka.MovementParameterFieldEnabled=True; IlfCommand=LIN
;ENDFOLD
$BWDSTART = FALSE
LDAT_ACT=LCPDATC296
FDAT_ACT=FC296
$ORI_TYPE = #VAR
$CIRC_TYPE = #PATH
BAS (#CP_PARAMS,0.1)
SET_CD_PARAMS (0)
CIRC XCAux296, XCDes296 C_DIS

;ENDFOLD
;FOLD LIN P297 CONT Vel=1 m/s CPDATP297 Tool[2] Base[10] ;%{PE}
;FOLD Parameters ;%{h}
;Params IlfProvider=kukaroboter.basistech.inlineforms.movement.old; Kuka.IsGlobalPoint=False; Kuka.PointName=P297; Kuka.BlendingEnabled=TRUE; Kuka.MoveDataName=CPDATP297; Kuka.VelocityPath=1; Kuka.CurrentCDSetIndex=0; Kuka.MovementParameterFieldEnabled=True; IlfCommand=LIN
;ENDFOLD
$BWDSTART = FALSE
LDAT_ACT=LCPDATP297
FDAT_ACT=FP297
BAS (#CP_PARAMS,1)
SET_CD_PARAMS (0)
LIN XP297 C_DIS

;ENDFOLD
;FOLD LIN P298 CONT Vel=1 m/s CPDATP298 Tool[2] Base[10] ;%{PE}
;FOLD Parameters ;%{h}
;Params IlfProvider=kukaroboter.basistech.inlineforms.movement.old; Kuka.IsGlobalPoint=False; Kuka.PointName=P298; Kuka.BlendingEnabled=TRUE; Kuka.MoveDataName=CPDATP298; Kuka.VelocityPath=1; Kuka.CurrentCDSetIndex=0; Kuka.MovementParameterFieldEnabled=True; IlfCommand=LIN
;ENDFOLD
$BWDSTART = FALSE
LDAT_ACT=LCPDATP298
FDAT_ACT=FP298
BAS (#CP_PARAMS,1)
SET_CD_PARAMS (0)
LIN XP298 C_DIS

;ENDFOLD
;FOLD CIRC CAux299 CDes299 CONT Vel=0.1 m/s CPDATC299 Tool[2] Base[10] ;%{PE}
;FOLD Parameters ;%{h}
;Params IlfProvider=kukaroboter.basistech.inlineforms.movement.old; Kuka.IsGlobalPoint=False; Kuka.PointName=CDes299; Kuka.BlendingEnabled=TRUE; Kuka.MoveDataName=CPDATC299; Kuka.VelocityPath=0.1; Kuka.CurrentCDSetIndex=0; Kuka.MovementParameterFieldEnabled=True; IlfCommand=LIN
;ENDFOLD
$BWDSTART = FALSE
LDAT_ACT=LCPDATC299
FDAT_ACT=FC299
$ORI_TYPE = #VAR
$CIRC_TYPE = #PATH
BAS (#CP_PARAMS,0.1)
SET_CD_PARAMS (0)
CIRC XCAux299, XCDes299 C_DIS

;ENDFOLD
;FOLD LIN P300 CONT Vel=1 m/s CPDATP300 Tool[2] Base[10] ;%{PE}
;FOLD Parameters ;%{h}
;Params IlfProvider=kukaroboter.basistech.inlineforms.movement.old; Kuka.IsGlobalPoint=False; Kuka.PointName=P300; Kuka.BlendingEnabled=TRUE; Kuka.MoveDataName=CPDATP300; Kuka.VelocityPath=1; Kuka.CurrentCDSetIndex=0; Kuka.MovementParameterFieldEnabled=True; IlfCommand=LIN
;ENDFOLD
$BWDSTART = FALSE
LDAT_ACT=LCPDATP300
FDAT_ACT=FP300
BAS (#CP_PARAMS,1)
SET_CD_PARAMS (0)
LIN XP300 C_DIS

;ENDFOLD
;FOLD LIN P301 CONT Vel=1 m/s CPDATP301 Tool[2] Base[10] ;%{PE}
;FOLD Parameters ;%{h}
;Params IlfProvider=kukaroboter.basistech.inlineforms.movement.old; Kuka.IsGlobalPoint=False; Kuka.PointName=P301; Kuka.BlendingEnabled=TRUE; Kuka.MoveDataName=CPDATP301; Kuka.VelocityPath=1; Kuka.CurrentCDSetIndex=0; Kuka.MovementParameterFieldEnabled=True; IlfCommand=LIN
;ENDFOLD
$BWDSTART = FALSE
LDAT_ACT=LCPDATP301
FDAT_ACT=FP301
BAS (#CP_PARAMS,1)
SET_CD_PARAMS (0)
LIN XP301 C_DIS

;ENDFOLD
;FOLD CIRC CAux302 CDes302 CONT Vel=0.1 m/s CPDATC302 Tool[2] Base[10] ;%{PE}
;FOLD Parameters ;%{h}
;Params IlfProvider=kukaroboter.basistech.inlineforms.movement.old; Kuka.IsGlobalPoint=False; Kuka.PointName=CDes302; Kuka.BlendingEnabled=TRUE; Kuka.MoveDataName=CPDATC302; Kuka.VelocityPath=0.1; Kuka.CurrentCDSetIndex=0; Kuka.MovementParameterFieldEnabled=True; IlfCommand=LIN
;ENDFOLD
$BWDSTART = FALSE
LDAT_ACT=LCPDATC302
FDAT_ACT=FC302
$ORI_TYPE = #VAR
$CIRC_TYPE = #PATH
BAS (#CP_PARAMS,0.1)
SET_CD_PARAMS (0)
CIRC XCAux302, XCDes302 C_DIS

;ENDFOLD
;FOLD LIN P303 CONT Vel=1 m/s CPDATP303 Tool[2] Base[10] ;%{PE}
;FOLD Parameters ;%{h}
;Params IlfProvider=kukaroboter.basistech.inlineforms.movement.old; Kuka.IsGlobalPoint=False; Kuka.PointName=P303; Kuka.BlendingEnabled=TRUE; Kuka.MoveDataName=CPDATP303; Kuka.VelocityPath=1; Kuka.CurrentCDSetIndex=0; Kuka.MovementParameterFieldEnabled=True; IlfCommand=LIN
;ENDFOLD
$BWDSTART = FALSE
LDAT_ACT=LCPDATP303
FDAT_ACT=FP303
BAS (#CP_PARAMS,1)
SET_CD_PARAMS (0)
LIN XP303 C_DIS

;ENDFOLD
;FOLD LIN P304 CONT Vel=1 m/s CPDATP304 Tool[2] Base[10] ;%{PE}
;FOLD Parameters ;%{h}
;Params IlfProvider=kukaroboter.basistech.inlineforms.movement.old; Kuka.IsGlobalPoint=False; Kuka.PointName=P304; Kuka.BlendingEnabled=TRUE; Kuka.MoveDataName=CPDATP304; Kuka.VelocityPath=1; Kuka.CurrentCDSetIndex=0; Kuka.MovementParameterFieldEnabled=True; IlfCommand=LIN
;ENDFOLD
$BWDSTART = FALSE
LDAT_ACT=LCPDATP304
FDAT_ACT=FP304
BAS (#CP_PARAMS,1)
SET_CD_PARAMS (0)
LIN XP304 C_DIS

;ENDFOLD
;FOLD CIRC CAux305 CDes305 CONT Vel=0.1 m/s CPDATC305 Tool[2] Base[10] ;%{PE}
;FOLD Parameters ;%{h}
;Params IlfProvider=kukaroboter.basistech.inlineforms.movement.old; Kuka.IsGlobalPoint=False; Kuka.PointName=CDes305; Kuka.BlendingEnabled=TRUE; Kuka.MoveDataName=CPDATC305; Kuka.VelocityPath=0.1; Kuka.CurrentCDSetIndex=0; Kuka.MovementParameterFieldEnabled=True; IlfCommand=LIN
;ENDFOLD
$BWDSTART = FALSE
LDAT_ACT=LCPDATC305
FDAT_ACT=FC305
$ORI_TYPE = #VAR
$CIRC_TYPE = #PATH
BAS (#CP_PARAMS,0.1)
SET_CD_PARAMS (0)
CIRC XCAux305, XCDes305 C_DIS

;ENDFOLD
;FOLD LIN P306 CONT Vel=1 m/s CPDATP306 Tool[2] Base[10] ;%{PE}
;FOLD Parameters ;%{h}
;Params IlfProvider=kukaroboter.basistech.inlineforms.movement.old; Kuka.IsGlobalPoint=False; Kuka.PointName=P306; Kuka.BlendingEnabled=TRUE; Kuka.MoveDataName=CPDATP306; Kuka.VelocityPath=1; Kuka.CurrentCDSetIndex=0; Kuka.MovementParameterFieldEnabled=True; IlfCommand=LIN
;ENDFOLD
$BWDSTART = FALSE
LDAT_ACT=LCPDATP306
FDAT_ACT=FP306
BAS (#CP_PARAMS,1)
SET_CD_PARAMS (0)
LIN XP306 C_DIS

;ENDFOLD
;FOLD LIN P307 CONT Vel=1 m/s CPDATP307 Tool[2] Base[10] ;%{PE}
;FOLD Parameters ;%{h}
;Params IlfProvider=kukaroboter.basistech.inlineforms.movement.old; Kuka.IsGlobalPoint=False; Kuka.PointName=P307; Kuka.BlendingEnabled=TRUE; Kuka.MoveDataName=CPDATP307; Kuka.VelocityPath=1; Kuka.CurrentCDSetIndex=0; Kuka.MovementParameterFieldEnabled=True; IlfCommand=LIN
;ENDFOLD
$BWDSTART = FALSE
LDAT_ACT=LCPDATP307
FDAT_ACT=FP307
BAS (#CP_PARAMS,1)
SET_CD_PARAMS (0)
LIN XP307 C_DIS

;ENDFOLD
;FOLD CIRC CAux308 CDes308 CONT Vel=0.1 m/s CPDATC308 Tool[2] Base[10] ;%{PE}
;FOLD Parameters ;%{h}
;Params IlfProvider=kukaroboter.basistech.inlineforms.movement.old; Kuka.IsGlobalPoint=False; Kuka.PointName=CDes308; Kuka.BlendingEnabled=TRUE; Kuka.MoveDataName=CPDATC308; Kuka.VelocityPath=0.1; Kuka.CurrentCDSetIndex=0; Kuka.MovementParameterFieldEnabled=True; IlfCommand=LIN
;ENDFOLD
$BWDSTART = FALSE
LDAT_ACT=LCPDATC308
FDAT_ACT=FC308
$ORI_TYPE = #VAR
$CIRC_TYPE = #PATH
BAS (#CP_PARAMS,0.1)
SET_CD_PARAMS (0)
CIRC XCAux308, XCDes308 C_DIS

;ENDFOLD
;FOLD LIN P309 CONT Vel=1 m/s CPDATP309 Tool[2] Base[10] ;%{PE}
;FOLD Parameters ;%{h}
;Params IlfProvider=kukaroboter.basistech.inlineforms.movement.old; Kuka.IsGlobalPoint=False; Kuka.PointName=P309; Kuka.BlendingEnabled=TRUE; Kuka.MoveDataName=CPDATP309; Kuka.VelocityPath=1; Kuka.CurrentCDSetIndex=0; Kuka.MovementParameterFieldEnabled=True; IlfCommand=LIN
;ENDFOLD
$BWDSTART = FALSE
LDAT_ACT=LCPDATP309
FDAT_ACT=FP309
BAS (#CP_PARAMS,1)
SET_CD_PARAMS (0)
LIN XP309 C_DIS

;ENDFOLD
;FOLD LIN P310 CONT Vel=1 m/s CPDATP310 Tool[2] Base[10] ;%{PE}
;FOLD Parameters ;%{h}
;Params IlfProvider=kukaroboter.basistech.inlineforms.movement.old; Kuka.IsGlobalPoint=False; Kuka.PointName=P310; Kuka.BlendingEnabled=TRUE; Kuka.MoveDataName=CPDATP310; Kuka.VelocityPath=1; Kuka.CurrentCDSetIndex=0; Kuka.MovementParameterFieldEnabled=True; IlfCommand=LIN
;ENDFOLD
$BWDSTART = FALSE
LDAT_ACT=LCPDATP310
FDAT_ACT=FP310
BAS (#CP_PARAMS,1)
SET_CD_PARAMS (0)
LIN XP310 C_DIS

;ENDFOLD
;FOLD CIRC CAux311 CDes311 CONT Vel=0.1 m/s CPDATC311 Tool[2] Base[10] ;%{PE}
;FOLD Parameters ;%{h}
;Params IlfProvider=kukaroboter.basistech.inlineforms.movement.old; Kuka.IsGlobalPoint=False; Kuka.PointName=CDes311; Kuka.BlendingEnabled=TRUE; Kuka.MoveDataName=CPDATC311; Kuka.VelocityPath=0.1; Kuka.CurrentCDSetIndex=0; Kuka.MovementParameterFieldEnabled=True; IlfCommand=LIN
;ENDFOLD
$BWDSTART = FALSE
LDAT_ACT=LCPDATC311
FDAT_ACT=FC311
$ORI_TYPE = #VAR
$CIRC_TYPE = #PATH
BAS (#CP_PARAMS,0.1)
SET_CD_PARAMS (0)
CIRC XCAux311, XCDes311 C_DIS

;ENDFOLD
;FOLD LIN P312 CONT Vel=1 m/s CPDATP312 Tool[2] Base[10] ;%{PE}
;FOLD Parameters ;%{h}
;Params IlfProvider=kukaroboter.basistech.inlineforms.movement.old; Kuka.IsGlobalPoint=False; Kuka.PointName=P312; Kuka.BlendingEnabled=TRUE; Kuka.MoveDataName=CPDATP312; Kuka.VelocityPath=1; Kuka.CurrentCDSetIndex=0; Kuka.MovementParameterFieldEnabled=True; IlfCommand=LIN
;ENDFOLD
$BWDSTART = FALSE
LDAT_ACT=LCPDATP312
FDAT_ACT=FP312
BAS (#CP_PARAMS,1)
SET_CD_PARAMS (0)
LIN XP312 C_DIS

;ENDFOLD
;FOLD LIN P313 CONT Vel=1 m/s CPDATP313 Tool[2] Base[10] ;%{PE}
;FOLD Parameters ;%{h}
;Params IlfProvider=kukaroboter.basistech.inlineforms.movement.old; Kuka.IsGlobalPoint=False; Kuka.PointName=P313; Kuka.BlendingEnabled=TRUE; Kuka.MoveDataName=CPDATP313; Kuka.VelocityPath=1; Kuka.CurrentCDSetIndex=0; Kuka.MovementParameterFieldEnabled=True; IlfCommand=LIN
;ENDFOLD
$BWDSTART = FALSE
LDAT_ACT=LCPDATP313
FDAT_ACT=FP313
BAS (#CP_PARAMS,1)
SET_CD_PARAMS (0)
LIN XP313 C_DIS

;ENDFOLD
;FOLD CIRC CAux314 CDes314 CONT Vel=0.1 m/s CPDATC314 Tool[2] Base[10] ;%{PE}
;FOLD Parameters ;%{h}
;Params IlfProvider=kukaroboter.basistech.inlineforms.movement.old; Kuka.IsGlobalPoint=False; Kuka.PointName=CDes314; Kuka.BlendingEnabled=TRUE; Kuka.MoveDataName=CPDATC314; Kuka.VelocityPath=0.1; Kuka.CurrentCDSetIndex=0; Kuka.MovementParameterFieldEnabled=True; IlfCommand=LIN
;ENDFOLD
$BWDSTART = FALSE
LDAT_ACT=LCPDATC314
FDAT_ACT=FC314
$ORI_TYPE = #VAR
$CIRC_TYPE = #PATH
BAS (#CP_PARAMS,0.1)
SET_CD_PARAMS (0)
CIRC XCAux314, XCDes314 C_DIS

;ENDFOLD
;FOLD LIN P315 CONT Vel=1 m/s CPDATP315 Tool[2] Base[10] ;%{PE}
;FOLD Parameters ;%{h}
;Params IlfProvider=kukaroboter.basistech.inlineforms.movement.old; Kuka.IsGlobalPoint=False; Kuka.PointName=P315; Kuka.BlendingEnabled=TRUE; Kuka.MoveDataName=CPDATP315; Kuka.VelocityPath=1; Kuka.CurrentCDSetIndex=0; Kuka.MovementParameterFieldEnabled=True; IlfCommand=LIN
;ENDFOLD
$BWDSTART = FALSE
LDAT_ACT=LCPDATP315
FDAT_ACT=FP315
BAS (#CP_PARAMS,1)
SET_CD_PARAMS (0)
LIN XP315 C_DIS

;ENDFOLD
;FOLD LIN P316 CONT Vel=1 m/s CPDATP316 Tool[2] Base[10] ;%{PE}
;FOLD Parameters ;%{h}
;Params IlfProvider=kukaroboter.basistech.inlineforms.movement.old; Kuka.IsGlobalPoint=False; Kuka.PointName=P316; Kuka.BlendingEnabled=TRUE; Kuka.MoveDataName=CPDATP316; Kuka.VelocityPath=1; Kuka.CurrentCDSetIndex=0; Kuka.MovementParameterFieldEnabled=True; IlfCommand=LIN
;ENDFOLD
$BWDSTART = FALSE
LDAT_ACT=LCPDATP316
FDAT_ACT=FP316
BAS (#CP_PARAMS,1)
SET_CD_PARAMS (0)
LIN XP316 C_DIS

;ENDFOLD
;FOLD CIRC CAux317 CDes317 CONT Vel=0.1 m/s CPDATC317 Tool[2] Base[10] ;%{PE}
;FOLD Parameters ;%{h}
;Params IlfProvider=kukaroboter.basistech.inlineforms.movement.old; Kuka.IsGlobalPoint=False; Kuka.PointName=CDes317; Kuka.BlendingEnabled=TRUE; Kuka.MoveDataName=CPDATC317; Kuka.VelocityPath=0.1; Kuka.CurrentCDSetIndex=0; Kuka.MovementParameterFieldEnabled=True; IlfCommand=LIN
;ENDFOLD
$BWDSTART = FALSE
LDAT_ACT=LCPDATC317
FDAT_ACT=FC317
$ORI_TYPE = #VAR
$CIRC_TYPE = #PATH
BAS (#CP_PARAMS,0.1)
SET_CD_PARAMS (0)
CIRC XCAux317, XCDes317 C_DIS

;ENDFOLD
;FOLD LIN P318 CONT Vel=1 m/s CPDATP318 Tool[2] Base[10] ;%{PE}
;FOLD Parameters ;%{h}
;Params IlfProvider=kukaroboter.basistech.inlineforms.movement.old; Kuka.IsGlobalPoint=False; Kuka.PointName=P318; Kuka.BlendingEnabled=TRUE; Kuka.MoveDataName=CPDATP318; Kuka.VelocityPath=1; Kuka.CurrentCDSetIndex=0; Kuka.MovementParameterFieldEnabled=True; IlfCommand=LIN
;ENDFOLD
$BWDSTART = FALSE
LDAT_ACT=LCPDATP318
FDAT_ACT=FP318
BAS (#CP_PARAMS,1)
SET_CD_PARAMS (0)
LIN XP318 C_DIS

;ENDFOLD
;FOLD LIN P319 CONT Vel=1 m/s CPDATP319 Tool[2] Base[10] ;%{PE}
;FOLD Parameters ;%{h}
;Params IlfProvider=kukaroboter.basistech.inlineforms.movement.old; Kuka.IsGlobalPoint=False; Kuka.PointName=P319; Kuka.BlendingEnabled=TRUE; Kuka.MoveDataName=CPDATP319; Kuka.VelocityPath=1; Kuka.CurrentCDSetIndex=0; Kuka.MovementParameterFieldEnabled=True; IlfCommand=LIN
;ENDFOLD
$BWDSTART = FALSE
LDAT_ACT=LCPDATP319
FDAT_ACT=FP319
BAS (#CP_PARAMS,1)
SET_CD_PARAMS (0)
LIN XP319 C_DIS

;ENDFOLD
;FOLD CIRC CAux320 CDes320 CONT Vel=0.1 m/s CPDATC320 Tool[2] Base[10] ;%{PE}
;FOLD Parameters ;%{h}
;Params IlfProvider=kukaroboter.basistech.inlineforms.movement.old; Kuka.IsGlobalPoint=False; Kuka.PointName=CDes320; Kuka.BlendingEnabled=TRUE; Kuka.MoveDataName=CPDATC320; Kuka.VelocityPath=0.1; Kuka.CurrentCDSetIndex=0; Kuka.MovementParameterFieldEnabled=True; IlfCommand=LIN
;ENDFOLD
$BWDSTART = FALSE
LDAT_ACT=LCPDATC320
FDAT_ACT=FC320
$ORI_TYPE = #VAR
$CIRC_TYPE = #PATH
BAS (#CP_PARAMS,0.1)
SET_CD_PARAMS (0)
CIRC XCAux320, XCDes320 C_DIS

;ENDFOLD
;FOLD LIN P321 CONT Vel=1 m/s CPDATP321 Tool[2] Base[10] ;%{PE}
;FOLD Parameters ;%{h}
;Params IlfProvider=kukaroboter.basistech.inlineforms.movement.old; Kuka.IsGlobalPoint=False; Kuka.PointName=P321; Kuka.BlendingEnabled=TRUE; Kuka.MoveDataName=CPDATP321; Kuka.VelocityPath=1; Kuka.CurrentCDSetIndex=0; Kuka.MovementParameterFieldEnabled=True; IlfCommand=LIN
;ENDFOLD
$BWDSTART = FALSE
LDAT_ACT=LCPDATP321
FDAT_ACT=FP321
BAS (#CP_PARAMS,1)
SET_CD_PARAMS (0)
LIN XP321 C_DIS

;ENDFOLD
;FOLD LIN P322 CONT Vel=1 m/s CPDATP322 Tool[2] Base[10] ;%{PE}
;FOLD Parameters ;%{h}
;Params IlfProvider=kukaroboter.basistech.inlineforms.movement.old; Kuka.IsGlobalPoint=False; Kuka.PointName=P322; Kuka.BlendingEnabled=TRUE; Kuka.MoveDataName=CPDATP322; Kuka.VelocityPath=1; Kuka.CurrentCDSetIndex=0; Kuka.MovementParameterFieldEnabled=True; IlfCommand=LIN
;ENDFOLD
$BWDSTART = FALSE
LDAT_ACT=LCPDATP322
FDAT_ACT=FP322
BAS (#CP_PARAMS,1)
SET_CD_PARAMS (0)
LIN XP322 C_DIS

;ENDFOLD
;FOLD CIRC CAux323 CDes323 CONT Vel=0.1 m/s CPDATC323 Tool[2] Base[10] ;%{PE}
;FOLD Parameters ;%{h}
;Params IlfProvider=kukaroboter.basistech.inlineforms.movement.old; Kuka.IsGlobalPoint=False; Kuka.PointName=CDes323; Kuka.BlendingEnabled=TRUE; Kuka.MoveDataName=CPDATC323; Kuka.VelocityPath=0.1; Kuka.CurrentCDSetIndex=0; Kuka.MovementParameterFieldEnabled=True; IlfCommand=LIN
;ENDFOLD
$BWDSTART = FALSE
LDAT_ACT=LCPDATC323
FDAT_ACT=FC323
$ORI_TYPE = #VAR
$CIRC_TYPE = #PATH
BAS (#CP_PARAMS,0.1)
SET_CD_PARAMS (0)
CIRC XCAux323, XCDes323 C_DIS

;ENDFOLD
;FOLD LIN P324 CONT Vel=1 m/s CPDATP324 Tool[2] Base[10] ;%{PE}
;FOLD Parameters ;%{h}
;Params IlfProvider=kukaroboter.basistech.inlineforms.movement.old; Kuka.IsGlobalPoint=False; Kuka.PointName=P324; Kuka.BlendingEnabled=TRUE; Kuka.MoveDataName=CPDATP324; Kuka.VelocityPath=1; Kuka.CurrentCDSetIndex=0; Kuka.MovementParameterFieldEnabled=True; IlfCommand=LIN
;ENDFOLD
$BWDSTART = FALSE
LDAT_ACT=LCPDATP324
FDAT_ACT=FP324
BAS (#CP_PARAMS,1)
SET_CD_PARAMS (0)
LIN XP324 C_DIS

;ENDFOLD
;FOLD LIN P325 CONT Vel=1 m/s CPDATP325 Tool[2] Base[10] ;%{PE}
;FOLD Parameters ;%{h}
;Params IlfProvider=kukaroboter.basistech.inlineforms.movement.old; Kuka.IsGlobalPoint=False; Kuka.PointName=P325; Kuka.BlendingEnabled=TRUE; Kuka.MoveDataName=CPDATP325; Kuka.VelocityPath=1; Kuka.CurrentCDSetIndex=0; Kuka.MovementParameterFieldEnabled=True; IlfCommand=LIN
;ENDFOLD
$BWDSTART = FALSE
LDAT_ACT=LCPDATP325
FDAT_ACT=FP325
BAS (#CP_PARAMS,1)
SET_CD_PARAMS (0)
LIN XP325 C_DIS

;ENDFOLD
;FOLD CIRC CAux326 CDes326 CONT Vel=0.1 m/s CPDATC326 Tool[2] Base[10] ;%{PE}
;FOLD Parameters ;%{h}
;Params IlfProvider=kukaroboter.basistech.inlineforms.movement.old; Kuka.IsGlobalPoint=False; Kuka.PointName=CDes326; Kuka.BlendingEnabled=TRUE; Kuka.MoveDataName=CPDATC326; Kuka.VelocityPath=0.1; Kuka.CurrentCDSetIndex=0; Kuka.MovementParameterFieldEnabled=True; IlfCommand=LIN
;ENDFOLD
$BWDSTART = FALSE
LDAT_ACT=LCPDATC326
FDAT_ACT=FC326
$ORI_TYPE = #VAR
$CIRC_TYPE = #PATH
BAS (#CP_PARAMS,0.1)
SET_CD_PARAMS (0)
CIRC XCAux326, XCDes326 C_DIS

;ENDFOLD
;FOLD LIN P327 CONT Vel=1 m/s CPDATP327 Tool[2] Base[10] ;%{PE}
;FOLD Parameters ;%{h}
;Params IlfProvider=kukaroboter.basistech.inlineforms.movement.old; Kuka.IsGlobalPoint=False; Kuka.PointName=P327; Kuka.BlendingEnabled=TRUE; Kuka.MoveDataName=CPDATP327; Kuka.VelocityPath=1; Kuka.CurrentCDSetIndex=0; Kuka.MovementParameterFieldEnabled=True; IlfCommand=LIN
;ENDFOLD
$BWDSTART = FALSE
LDAT_ACT=LCPDATP327
FDAT_ACT=FP327
BAS (#CP_PARAMS,1)
SET_CD_PARAMS (0)
LIN XP327 C_DIS

;ENDFOLD
;FOLD LIN P328 CONT Vel=1 m/s CPDATP328 Tool[2] Base[10] ;%{PE}
;FOLD Parameters ;%{h}
;Params IlfProvider=kukaroboter.basistech.inlineforms.movement.old; Kuka.IsGlobalPoint=False; Kuka.PointName=P328; Kuka.BlendingEnabled=TRUE; Kuka.MoveDataName=CPDATP328; Kuka.VelocityPath=1; Kuka.CurrentCDSetIndex=0; Kuka.MovementParameterFieldEnabled=True; IlfCommand=LIN
;ENDFOLD
$BWDSTART = FALSE
LDAT_ACT=LCPDATP328
FDAT_ACT=FP328
BAS (#CP_PARAMS,1)
SET_CD_PARAMS (0)
LIN XP328 C_DIS

;ENDFOLD
;FOLD CIRC CAux329 CDes329 CONT Vel=0.1 m/s CPDATC329 Tool[2] Base[10] ;%{PE}
;FOLD Parameters ;%{h}
;Params IlfProvider=kukaroboter.basistech.inlineforms.movement.old; Kuka.IsGlobalPoint=False; Kuka.PointName=CDes329; Kuka.BlendingEnabled=TRUE; Kuka.MoveDataName=CPDATC329; Kuka.VelocityPath=0.1; Kuka.CurrentCDSetIndex=0; Kuka.MovementParameterFieldEnabled=True; IlfCommand=LIN
;ENDFOLD
$BWDSTART = FALSE
LDAT_ACT=LCPDATC329
FDAT_ACT=FC329
$ORI_TYPE = #VAR
$CIRC_TYPE = #PATH
BAS (#CP_PARAMS,0.1)
SET_CD_PARAMS (0)
CIRC XCAux329, XCDes329 C_DIS

;ENDFOLD
;FOLD LIN P330 CONT Vel=1 m/s CPDATP330 Tool[2] Base[10] ;%{PE}
;FOLD Parameters ;%{h}
;Params IlfProvider=kukaroboter.basistech.inlineforms.movement.old; Kuka.IsGlobalPoint=False; Kuka.PointName=P330; Kuka.BlendingEnabled=TRUE; Kuka.MoveDataName=CPDATP330; Kuka.VelocityPath=1; Kuka.CurrentCDSetIndex=0; Kuka.MovementParameterFieldEnabled=True; IlfCommand=LIN
;ENDFOLD
$BWDSTART = FALSE
LDAT_ACT=LCPDATP330
FDAT_ACT=FP330
BAS (#CP_PARAMS,1)
SET_CD_PARAMS (0)
LIN XP330 C_DIS

;ENDFOLD
;FOLD LIN P331 CONT Vel=1 m/s CPDATP331 Tool[2] Base[10] ;%{PE}
;FOLD Parameters ;%{h}
;Params IlfProvider=kukaroboter.basistech.inlineforms.movement.old; Kuka.IsGlobalPoint=False; Kuka.PointName=P331; Kuka.BlendingEnabled=TRUE; Kuka.MoveDataName=CPDATP331; Kuka.VelocityPath=1; Kuka.CurrentCDSetIndex=0; Kuka.MovementParameterFieldEnabled=True; IlfCommand=LIN
;ENDFOLD
$BWDSTART = FALSE
LDAT_ACT=LCPDATP331
FDAT_ACT=FP331
BAS (#CP_PARAMS,1)
SET_CD_PARAMS (0)
LIN XP331 C_DIS

;ENDFOLD
;FOLD CIRC CAux332 CDes332 CONT Vel=0.1 m/s CPDATC332 Tool[2] Base[10] ;%{PE}
;FOLD Parameters ;%{h}
;Params IlfProvider=kukaroboter.basistech.inlineforms.movement.old; Kuka.IsGlobalPoint=False; Kuka.PointName=CDes332; Kuka.BlendingEnabled=TRUE; Kuka.MoveDataName=CPDATC332; Kuka.VelocityPath=0.1; Kuka.CurrentCDSetIndex=0; Kuka.MovementParameterFieldEnabled=True; IlfCommand=LIN
;ENDFOLD
$BWDSTART = FALSE
LDAT_ACT=LCPDATC332
FDAT_ACT=FC332
$ORI_TYPE = #VAR
$CIRC_TYPE = #PATH
BAS (#CP_PARAMS,0.1)
SET_CD_PARAMS (0)
CIRC XCAux332, XCDes332 C_DIS

;ENDFOLD
;FOLD LIN P333 CONT Vel=1 m/s CPDATP333 Tool[2] Base[10] ;%{PE}
;FOLD Parameters ;%{h}
;Params IlfProvider=kukaroboter.basistech.inlineforms.movement.old; Kuka.IsGlobalPoint=False; Kuka.PointName=P333; Kuka.BlendingEnabled=TRUE; Kuka.MoveDataName=CPDATP333; Kuka.VelocityPath=1; Kuka.CurrentCDSetIndex=0; Kuka.MovementParameterFieldEnabled=True; IlfCommand=LIN
;ENDFOLD
$BWDSTART = FALSE
LDAT_ACT=LCPDATP333
FDAT_ACT=FP333
BAS (#CP_PARAMS,1)
SET_CD_PARAMS (0)
LIN XP333 C_DIS

;ENDFOLD
;FOLD LIN P334 CONT Vel=1 m/s CPDATP334 Tool[2] Base[10] ;%{PE}
;FOLD Parameters ;%{h}
;Params IlfProvider=kukaroboter.basistech.inlineforms.movement.old; Kuka.IsGlobalPoint=False; Kuka.PointName=P334; Kuka.BlendingEnabled=TRUE; Kuka.MoveDataName=CPDATP334; Kuka.VelocityPath=1; Kuka.CurrentCDSetIndex=0; Kuka.MovementParameterFieldEnabled=True; IlfCommand=LIN
;ENDFOLD
$BWDSTART = FALSE
LDAT_ACT=LCPDATP334
FDAT_ACT=FP334
BAS (#CP_PARAMS,1)
SET_CD_PARAMS (0)
LIN XP334 C_DIS

;ENDFOLD
;FOLD CIRC CAux335 CDes335 CONT Vel=0.1 m/s CPDATC335 Tool[2] Base[10] ;%{PE}
;FOLD Parameters ;%{h}
;Params IlfProvider=kukaroboter.basistech.inlineforms.movement.old; Kuka.IsGlobalPoint=False; Kuka.PointName=CDes335; Kuka.BlendingEnabled=TRUE; Kuka.MoveDataName=CPDATC335; Kuka.VelocityPath=0.1; Kuka.CurrentCDSetIndex=0; Kuka.MovementParameterFieldEnabled=True; IlfCommand=LIN
;ENDFOLD
$BWDSTART = FALSE
LDAT_ACT=LCPDATC335
FDAT_ACT=FC335
$ORI_TYPE = #VAR
$CIRC_TYPE = #PATH
BAS (#CP_PARAMS,0.1)
SET_CD_PARAMS (0)
CIRC XCAux335, XCDes335 C_DIS

;ENDFOLD
;FOLD LIN P336 CONT Vel=1 m/s CPDATP336 Tool[2] Base[10] ;%{PE}
;FOLD Parameters ;%{h}
;Params IlfProvider=kukaroboter.basistech.inlineforms.movement.old; Kuka.IsGlobalPoint=False; Kuka.PointName=P336; Kuka.BlendingEnabled=TRUE; Kuka.MoveDataName=CPDATP336; Kuka.VelocityPath=1; Kuka.CurrentCDSetIndex=0; Kuka.MovementParameterFieldEnabled=True; IlfCommand=LIN
;ENDFOLD
$BWDSTART = FALSE
LDAT_ACT=LCPDATP336
FDAT_ACT=FP336
BAS (#CP_PARAMS,1)
SET_CD_PARAMS (0)
LIN XP336 C_DIS

;ENDFOLD
;FOLD LIN P337 CONT Vel=1 m/s CPDATP337 Tool[2] Base[10] ;%{PE}
;FOLD Parameters ;%{h}
;Params IlfProvider=kukaroboter.basistech.inlineforms.movement.old; Kuka.IsGlobalPoint=False; Kuka.PointName=P337; Kuka.BlendingEnabled=TRUE; Kuka.MoveDataName=CPDATP337; Kuka.VelocityPath=1; Kuka.CurrentCDSetIndex=0; Kuka.MovementParameterFieldEnabled=True; IlfCommand=LIN
;ENDFOLD
$BWDSTART = FALSE
LDAT_ACT=LCPDATP337
FDAT_ACT=FP337
BAS (#CP_PARAMS,1)
SET_CD_PARAMS (0)
LIN XP337 C_DIS

;ENDFOLD
;FOLD CIRC CAux338 CDes338 CONT Vel=0.1 m/s CPDATC338 Tool[2] Base[10] ;%{PE}
;FOLD Parameters ;%{h}
;Params IlfProvider=kukaroboter.basistech.inlineforms.movement.old; Kuka.IsGlobalPoint=False; Kuka.PointName=CDes338; Kuka.BlendingEnabled=TRUE; Kuka.MoveDataName=CPDATC338; Kuka.VelocityPath=0.1; Kuka.CurrentCDSetIndex=0; Kuka.MovementParameterFieldEnabled=True; IlfCommand=LIN
;ENDFOLD
$BWDSTART = FALSE
LDAT_ACT=LCPDATC338
FDAT_ACT=FC338
$ORI_TYPE = #VAR
$CIRC_TYPE = #PATH
BAS (#CP_PARAMS,0.1)
SET_CD_PARAMS (0)
CIRC XCAux338, XCDes338 C_DIS

;ENDFOLD
;FOLD LIN P339 CONT Vel=1 m/s CPDATP339 Tool[2] Base[10] ;%{PE}
;FOLD Parameters ;%{h}
;Params IlfProvider=kukaroboter.basistech.inlineforms.movement.old; Kuka.IsGlobalPoint=False; Kuka.PointName=P339; Kuka.BlendingEnabled=TRUE; Kuka.MoveDataName=CPDATP339; Kuka.VelocityPath=1; Kuka.CurrentCDSetIndex=0; Kuka.MovementParameterFieldEnabled=True; IlfCommand=LIN
;ENDFOLD
$BWDSTART = FALSE
LDAT_ACT=LCPDATP339
FDAT_ACT=FP339
BAS (#CP_PARAMS,1)
SET_CD_PARAMS (0)
LIN XP339 C_DIS

;ENDFOLD
;FOLD LIN P340 CONT Vel=1 m/s CPDATP340 Tool[2] Base[10] ;%{PE}
;FOLD Parameters ;%{h}
;Params IlfProvider=kukaroboter.basistech.inlineforms.movement.old; Kuka.IsGlobalPoint=False; Kuka.PointName=P340; Kuka.BlendingEnabled=TRUE; Kuka.MoveDataName=CPDATP340; Kuka.VelocityPath=1; Kuka.CurrentCDSetIndex=0; Kuka.MovementParameterFieldEnabled=True; IlfCommand=LIN
;ENDFOLD
$BWDSTART = FALSE
LDAT_ACT=LCPDATP340
FDAT_ACT=FP340
BAS (#CP_PARAMS,1)
SET_CD_PARAMS (0)
LIN XP340 C_DIS

;ENDFOLD
;FOLD CIRC CAux341 CDes341 CONT Vel=0.1 m/s CPDATC341 Tool[2] Base[10] ;%{PE}
;FOLD Parameters ;%{h}
;Params IlfProvider=kukaroboter.basistech.inlineforms.movement.old; Kuka.IsGlobalPoint=False; Kuka.PointName=CDes341; Kuka.BlendingEnabled=TRUE; Kuka.MoveDataName=CPDATC341; Kuka.VelocityPath=0.1; Kuka.CurrentCDSetIndex=0; Kuka.MovementParameterFieldEnabled=True; IlfCommand=LIN
;ENDFOLD
$BWDSTART = FALSE
LDAT_ACT=LCPDATC341
FDAT_ACT=FC341
$ORI_TYPE = #VAR
$CIRC_TYPE = #PATH
BAS (#CP_PARAMS,0.1)
SET_CD_PARAMS (0)
CIRC XCAux341, XCDes341 C_DIS

;ENDFOLD
;FOLD LIN P342 CONT Vel=1 m/s CPDATP342 Tool[2] Base[10] ;%{PE}
;FOLD Parameters ;%{h}
;Params IlfProvider=kukaroboter.basistech.inlineforms.movement.old; Kuka.IsGlobalPoint=False; Kuka.PointName=P342; Kuka.BlendingEnabled=TRUE; Kuka.MoveDataName=CPDATP342; Kuka.VelocityPath=1; Kuka.CurrentCDSetIndex=0; Kuka.MovementParameterFieldEnabled=True; IlfCommand=LIN
;ENDFOLD
$BWDSTART = FALSE
LDAT_ACT=LCPDATP342
FDAT_ACT=FP342
BAS (#CP_PARAMS,1)
SET_CD_PARAMS (0)
LIN XP342 C_DIS

;ENDFOLD
;FOLD LIN P343 CONT Vel=1 m/s CPDATP343 Tool[2] Base[10] ;%{PE}
;FOLD Parameters ;%{h}
;Params IlfProvider=kukaroboter.basistech.inlineforms.movement.old; Kuka.IsGlobalPoint=False; Kuka.PointName=P343; Kuka.BlendingEnabled=TRUE; Kuka.MoveDataName=CPDATP343; Kuka.VelocityPath=1; Kuka.CurrentCDSetIndex=0; Kuka.MovementParameterFieldEnabled=True; IlfCommand=LIN
;ENDFOLD
$BWDSTART = FALSE
LDAT_ACT=LCPDATP343
FDAT_ACT=FP343
BAS (#CP_PARAMS,1)
SET_CD_PARAMS (0)
LIN XP343 C_DIS

;ENDFOLD
;FOLD CIRC CAux344 CDes344 CONT Vel=0.1 m/s CPDATC344 Tool[2] Base[10] ;%{PE}
;FOLD Parameters ;%{h}
;Params IlfProvider=kukaroboter.basistech.inlineforms.movement.old; Kuka.IsGlobalPoint=False; Kuka.PointName=CDes344; Kuka.BlendingEnabled=TRUE; Kuka.MoveDataName=CPDATC344; Kuka.VelocityPath=0.1; Kuka.CurrentCDSetIndex=0; Kuka.MovementParameterFieldEnabled=True; IlfCommand=LIN
;ENDFOLD
$BWDSTART = FALSE
LDAT_ACT=LCPDATC344
FDAT_ACT=FC344
$ORI_TYPE = #VAR
$CIRC_TYPE = #PATH
BAS (#CP_PARAMS,0.1)
SET_CD_PARAMS (0)
CIRC XCAux344, XCDes344 C_DIS

;ENDFOLD
;FOLD LIN P345 CONT Vel=1 m/s CPDATP345 Tool[2] Base[10] ;%{PE}
;FOLD Parameters ;%{h}
;Params IlfProvider=kukaroboter.basistech.inlineforms.movement.old; Kuka.IsGlobalPoint=False; Kuka.PointName=P345; Kuka.BlendingEnabled=TRUE; Kuka.MoveDataName=CPDATP345; Kuka.VelocityPath=1; Kuka.CurrentCDSetIndex=0; Kuka.MovementParameterFieldEnabled=True; IlfCommand=LIN
;ENDFOLD
$BWDSTART = FALSE
LDAT_ACT=LCPDATP345
FDAT_ACT=FP345
BAS (#CP_PARAMS,1)
SET_CD_PARAMS (0)
LIN XP345 C_DIS

;ENDFOLD
;FOLD LIN P346 CONT Vel=1 m/s CPDATP346 Tool[2] Base[10] ;%{PE}
;FOLD Parameters ;%{h}
;Params IlfProvider=kukaroboter.basistech.inlineforms.movement.old; Kuka.IsGlobalPoint=False; Kuka.PointName=P346; Kuka.BlendingEnabled=TRUE; Kuka.MoveDataName=CPDATP346; Kuka.VelocityPath=1; Kuka.CurrentCDSetIndex=0; Kuka.MovementParameterFieldEnabled=True; IlfCommand=LIN
;ENDFOLD
$BWDSTART = FALSE
LDAT_ACT=LCPDATP346
FDAT_ACT=FP346
BAS (#CP_PARAMS,1)
SET_CD_PARAMS (0)
LIN XP346 C_DIS

;ENDFOLD
;FOLD CIRC CAux347 CDes347 CONT Vel=0.1 m/s CPDATC347 Tool[2] Base[10] ;%{PE}
;FOLD Parameters ;%{h}
;Params IlfProvider=kukaroboter.basistech.inlineforms.movement.old; Kuka.IsGlobalPoint=False; Kuka.PointName=CDes347; Kuka.BlendingEnabled=TRUE; Kuka.MoveDataName=CPDATC347; Kuka.VelocityPath=0.1; Kuka.CurrentCDSetIndex=0; Kuka.MovementParameterFieldEnabled=True; IlfCommand=LIN
;ENDFOLD
$BWDSTART = FALSE
LDAT_ACT=LCPDATC347
FDAT_ACT=FC347
$ORI_TYPE = #VAR
$CIRC_TYPE = #PATH
BAS (#CP_PARAMS,0.1)
SET_CD_PARAMS (0)
CIRC XCAux347, XCDes347 C_DIS

;ENDFOLD
;FOLD LIN P348 CONT Vel=1 m/s CPDATP348 Tool[2] Base[10] ;%{PE}
;FOLD Parameters ;%{h}
;Params IlfProvider=kukaroboter.basistech.inlineforms.movement.old; Kuka.IsGlobalPoint=False; Kuka.PointName=P348; Kuka.BlendingEnabled=TRUE; Kuka.MoveDataName=CPDATP348; Kuka.VelocityPath=1; Kuka.CurrentCDSetIndex=0; Kuka.MovementParameterFieldEnabled=True; IlfCommand=LIN
;ENDFOLD
$BWDSTART = FALSE
LDAT_ACT=LCPDATP348
FDAT_ACT=FP348
BAS (#CP_PARAMS,1)
SET_CD_PARAMS (0)
LIN XP348 C_DIS

;ENDFOLD
;FOLD LIN P349 CONT Vel=1 m/s CPDATP349 Tool[2] Base[10] ;%{PE}
;FOLD Parameters ;%{h}
;Params IlfProvider=kukaroboter.basistech.inlineforms.movement.old; Kuka.IsGlobalPoint=False; Kuka.PointName=P349; Kuka.BlendingEnabled=TRUE; Kuka.MoveDataName=CPDATP349; Kuka.VelocityPath=1; Kuka.CurrentCDSetIndex=0; Kuka.MovementParameterFieldEnabled=True; IlfCommand=LIN
;ENDFOLD
$BWDSTART = FALSE
LDAT_ACT=LCPDATP349
FDAT_ACT=FP349
BAS (#CP_PARAMS,1)
SET_CD_PARAMS (0)
LIN XP349 C_DIS

;ENDFOLD
;FOLD CIRC CAux350 CDes350 CONT Vel=0.1 m/s CPDATC350 Tool[2] Base[10] ;%{PE}
;FOLD Parameters ;%{h}
;Params IlfProvider=kukaroboter.basistech.inlineforms.movement.old; Kuka.IsGlobalPoint=False; Kuka.PointName=CDes350; Kuka.BlendingEnabled=TRUE; Kuka.MoveDataName=CPDATC350; Kuka.VelocityPath=0.1; Kuka.CurrentCDSetIndex=0; Kuka.MovementParameterFieldEnabled=True; IlfCommand=LIN
;ENDFOLD
$BWDSTART = FALSE
LDAT_ACT=LCPDATC350
FDAT_ACT=FC350
$ORI_TYPE = #VAR
$CIRC_TYPE = #PATH
BAS (#CP_PARAMS,0.1)
SET_CD_PARAMS (0)
CIRC XCAux350, XCDes350 C_DIS

;ENDFOLD
;FOLD LIN P351 CONT Vel=1 m/s CPDATP351 Tool[2] Base[10] ;%{PE}
;FOLD Parameters ;%{h}
;Params IlfProvider=kukaroboter.basistech.inlineforms.movement.old; Kuka.IsGlobalPoint=False; Kuka.PointName=P351; Kuka.BlendingEnabled=TRUE; Kuka.MoveDataName=CPDATP351; Kuka.VelocityPath=1; Kuka.CurrentCDSetIndex=0; Kuka.MovementParameterFieldEnabled=True; IlfCommand=LIN
;ENDFOLD
$BWDSTART = FALSE
LDAT_ACT=LCPDATP351
FDAT_ACT=FP351
BAS (#CP_PARAMS,1)
SET_CD_PARAMS (0)
LIN XP351 C_DIS

;ENDFOLD
;FOLD LIN P352 CONT Vel=1 m/s CPDATP352 Tool[2] Base[10] ;%{PE}
;FOLD Parameters ;%{h}
;Params IlfProvider=kukaroboter.basistech.inlineforms.movement.old; Kuka.IsGlobalPoint=False; Kuka.PointName=P352; Kuka.BlendingEnabled=TRUE; Kuka.MoveDataName=CPDATP352; Kuka.VelocityPath=1; Kuka.CurrentCDSetIndex=0; Kuka.MovementParameterFieldEnabled=True; IlfCommand=LIN
;ENDFOLD
$BWDSTART = FALSE
LDAT_ACT=LCPDATP352
FDAT_ACT=FP352
BAS (#CP_PARAMS,1)
SET_CD_PARAMS (0)
LIN XP352 C_DIS

;ENDFOLD
;FOLD CIRC CAux353 CDes353 CONT Vel=0.1 m/s CPDATC353 Tool[2] Base[10] ;%{PE}
;FOLD Parameters ;%{h}
;Params IlfProvider=kukaroboter.basistech.inlineforms.movement.old; Kuka.IsGlobalPoint=False; Kuka.PointName=CDes353; Kuka.BlendingEnabled=TRUE; Kuka.MoveDataName=CPDATC353; Kuka.VelocityPath=0.1; Kuka.CurrentCDSetIndex=0; Kuka.MovementParameterFieldEnabled=True; IlfCommand=LIN
;ENDFOLD
$BWDSTART = FALSE
LDAT_ACT=LCPDATC353
FDAT_ACT=FC353
$ORI_TYPE = #VAR
$CIRC_TYPE = #PATH
BAS (#CP_PARAMS,0.1)
SET_CD_PARAMS (0)
CIRC XCAux353, XCDes353 C_DIS

;ENDFOLD
;FOLD LIN P354 CONT Vel=1 m/s CPDATP354 Tool[2] Base[10] ;%{PE}
;FOLD Parameters ;%{h}
;Params IlfProvider=kukaroboter.basistech.inlineforms.movement.old; Kuka.IsGlobalPoint=False; Kuka.PointName=P354; Kuka.BlendingEnabled=TRUE; Kuka.MoveDataName=CPDATP354; Kuka.VelocityPath=1; Kuka.CurrentCDSetIndex=0; Kuka.MovementParameterFieldEnabled=True; IlfCommand=LIN
;ENDFOLD
$BWDSTART = FALSE
LDAT_ACT=LCPDATP354
FDAT_ACT=FP354
BAS (#CP_PARAMS,1)
SET_CD_PARAMS (0)
LIN XP354 C_DIS

;ENDFOLD
;FOLD LIN P355 CONT Vel=1 m/s CPDATP355 Tool[2] Base[10] ;%{PE}
;FOLD Parameters ;%{h}
;Params IlfProvider=kukaroboter.basistech.inlineforms.movement.old; Kuka.IsGlobalPoint=False; Kuka.PointName=P355; Kuka.BlendingEnabled=TRUE; Kuka.MoveDataName=CPDATP355; Kuka.VelocityPath=1; Kuka.CurrentCDSetIndex=0; Kuka.MovementParameterFieldEnabled=True; IlfCommand=LIN
;ENDFOLD
$BWDSTART = FALSE
LDAT_ACT=LCPDATP355
FDAT_ACT=FP355
BAS (#CP_PARAMS,1)
SET_CD_PARAMS (0)
LIN XP355 C_DIS

;ENDFOLD
;FOLD CIRC CAux356 CDes356 CONT Vel=0.1 m/s CPDATC356 Tool[2] Base[10] ;%{PE}
;FOLD Parameters ;%{h}
;Params IlfProvider=kukaroboter.basistech.inlineforms.movement.old; Kuka.IsGlobalPoint=False; Kuka.PointName=CDes356; Kuka.BlendingEnabled=TRUE; Kuka.MoveDataName=CPDATC356; Kuka.VelocityPath=0.1; Kuka.CurrentCDSetIndex=0; Kuka.MovementParameterFieldEnabled=True; IlfCommand=LIN
;ENDFOLD
$BWDSTART = FALSE
LDAT_ACT=LCPDATC356
FDAT_ACT=FC356
$ORI_TYPE = #VAR
$CIRC_TYPE = #PATH
BAS (#CP_PARAMS,0.1)
SET_CD_PARAMS (0)
CIRC XCAux356, XCDes356 C_DIS

;ENDFOLD
;FOLD LIN P357 CONT Vel=1 m/s CPDATP357 Tool[2] Base[10] ;%{PE}
;FOLD Parameters ;%{h}
;Params IlfProvider=kukaroboter.basistech.inlineforms.movement.old; Kuka.IsGlobalPoint=False; Kuka.PointName=P357; Kuka.BlendingEnabled=TRUE; Kuka.MoveDataName=CPDATP357; Kuka.VelocityPath=1; Kuka.CurrentCDSetIndex=0; Kuka.MovementParameterFieldEnabled=True; IlfCommand=LIN
;ENDFOLD
$BWDSTART = FALSE
LDAT_ACT=LCPDATP357
FDAT_ACT=FP357
BAS (#CP_PARAMS,1)
SET_CD_PARAMS (0)
LIN XP357 C_DIS

;ENDFOLD
;FOLD LIN P358 CONT Vel=1 m/s CPDATP358 Tool[2] Base[10] ;%{PE}
;FOLD Parameters ;%{h}
;Params IlfProvider=kukaroboter.basistech.inlineforms.movement.old; Kuka.IsGlobalPoint=False; Kuka.PointName=P358; Kuka.BlendingEnabled=TRUE; Kuka.MoveDataName=CPDATP358; Kuka.VelocityPath=1; Kuka.CurrentCDSetIndex=0; Kuka.MovementParameterFieldEnabled=True; IlfCommand=LIN
;ENDFOLD
$BWDSTART = FALSE
LDAT_ACT=LCPDATP358
FDAT_ACT=FP358
BAS (#CP_PARAMS,1)
SET_CD_PARAMS (0)
LIN XP358 C_DIS

;ENDFOLD
;FOLD CIRC CAux359 CDes359 CONT Vel=0.1 m/s CPDATC359 Tool[2] Base[10] ;%{PE}
;FOLD Parameters ;%{h}
;Params IlfProvider=kukaroboter.basistech.inlineforms.movement.old; Kuka.IsGlobalPoint=False; Kuka.PointName=CDes359; Kuka.BlendingEnabled=TRUE; Kuka.MoveDataName=CPDATC359; Kuka.VelocityPath=0.1; Kuka.CurrentCDSetIndex=0; Kuka.MovementParameterFieldEnabled=True; IlfCommand=LIN
;ENDFOLD
$BWDSTART = FALSE
LDAT_ACT=LCPDATC359
FDAT_ACT=FC359
$ORI_TYPE = #VAR
$CIRC_TYPE = #PATH
BAS (#CP_PARAMS,0.1)
SET_CD_PARAMS (0)
CIRC XCAux359, XCDes359 C_DIS

;ENDFOLD
;FOLD LIN P360 CONT Vel=1 m/s CPDATP360 Tool[2] Base[10] ;%{PE}
;FOLD Parameters ;%{h}
;Params IlfProvider=kukaroboter.basistech.inlineforms.movement.old; Kuka.IsGlobalPoint=False; Kuka.PointName=P360; Kuka.BlendingEnabled=TRUE; Kuka.MoveDataName=CPDATP360; Kuka.VelocityPath=1; Kuka.CurrentCDSetIndex=0; Kuka.MovementParameterFieldEnabled=True; IlfCommand=LIN
;ENDFOLD
$BWDSTART = FALSE
LDAT_ACT=LCPDATP360
FDAT_ACT=FP360
BAS (#CP_PARAMS,1)
SET_CD_PARAMS (0)
LIN XP360 C_DIS

;ENDFOLD
;FOLD LIN P361 CONT Vel=1 m/s CPDATP361 Tool[2] Base[10] ;%{PE}
;FOLD Parameters ;%{h}
;Params IlfProvider=kukaroboter.basistech.inlineforms.movement.old; Kuka.IsGlobalPoint=False; Kuka.PointName=P361; Kuka.BlendingEnabled=TRUE; Kuka.MoveDataName=CPDATP361; Kuka.VelocityPath=1; Kuka.CurrentCDSetIndex=0; Kuka.MovementParameterFieldEnabled=True; IlfCommand=LIN
;ENDFOLD
$BWDSTART = FALSE
LDAT_ACT=LCPDATP361
FDAT_ACT=FP361
BAS (#CP_PARAMS,1)
SET_CD_PARAMS (0)
LIN XP361 C_DIS

;ENDFOLD
;FOLD CIRC CAux362 CDes362 CONT Vel=0.1 m/s CPDATC362 Tool[2] Base[10] ;%{PE}
;FOLD Parameters ;%{h}
;Params IlfProvider=kukaroboter.basistech.inlineforms.movement.old; Kuka.IsGlobalPoint=False; Kuka.PointName=CDes362; Kuka.BlendingEnabled=TRUE; Kuka.MoveDataName=CPDATC362; Kuka.VelocityPath=0.1; Kuka.CurrentCDSetIndex=0; Kuka.MovementParameterFieldEnabled=True; IlfCommand=LIN
;ENDFOLD
$BWDSTART = FALSE
LDAT_ACT=LCPDATC362
FDAT_ACT=FC362
$ORI_TYPE = #VAR
$CIRC_TYPE = #PATH
BAS (#CP_PARAMS,0.1)
SET_CD_PARAMS (0)
CIRC XCAux362, XCDes362 C_DIS

;ENDFOLD
;FOLD LIN P363 CONT Vel=1 m/s CPDATP363 Tool[2] Base[10] ;%{PE}
;FOLD Parameters ;%{h}
;Params IlfProvider=kukaroboter.basistech.inlineforms.movement.old; Kuka.IsGlobalPoint=False; Kuka.PointName=P363; Kuka.BlendingEnabled=TRUE; Kuka.MoveDataName=CPDATP363; Kuka.VelocityPath=1; Kuka.CurrentCDSetIndex=0; Kuka.MovementParameterFieldEnabled=True; IlfCommand=LIN
;ENDFOLD
$BWDSTART = FALSE
LDAT_ACT=LCPDATP363
FDAT_ACT=FP363
BAS (#CP_PARAMS,1)
SET_CD_PARAMS (0)
LIN XP363 C_DIS

;ENDFOLD
;FOLD LIN P364 CONT Vel=1 m/s CPDATP364 Tool[2] Base[10] ;%{PE}
;FOLD Parameters ;%{h}
;Params IlfProvider=kukaroboter.basistech.inlineforms.movement.old; Kuka.IsGlobalPoint=False; Kuka.PointName=P364; Kuka.BlendingEnabled=TRUE; Kuka.MoveDataName=CPDATP364; Kuka.VelocityPath=1; Kuka.CurrentCDSetIndex=0; Kuka.MovementParameterFieldEnabled=True; IlfCommand=LIN
;ENDFOLD
$BWDSTART = FALSE
LDAT_ACT=LCPDATP364
FDAT_ACT=FP364
BAS (#CP_PARAMS,1)
SET_CD_PARAMS (0)
LIN XP364 C_DIS

;ENDFOLD
;FOLD CIRC CAux365 CDes365 CONT Vel=0.1 m/s CPDATC365 Tool[2] Base[10] ;%{PE}
;FOLD Parameters ;%{h}
;Params IlfProvider=kukaroboter.basistech.inlineforms.movement.old; Kuka.IsGlobalPoint=False; Kuka.PointName=CDes365; Kuka.BlendingEnabled=TRUE; Kuka.MoveDataName=CPDATC365; Kuka.VelocityPath=0.1; Kuka.CurrentCDSetIndex=0; Kuka.MovementParameterFieldEnabled=True; IlfCommand=LIN
;ENDFOLD
$BWDSTART = FALSE
LDAT_ACT=LCPDATC365
FDAT_ACT=FC365
$ORI_TYPE = #VAR
$CIRC_TYPE = #PATH
BAS (#CP_PARAMS,0.1)
SET_CD_PARAMS (0)
CIRC XCAux365, XCDes365 C_DIS

;ENDFOLD
;FOLD LIN P366 CONT Vel=1 m/s CPDATP366 Tool[2] Base[10] ;%{PE}
;FOLD Parameters ;%{h}
;Params IlfProvider=kukaroboter.basistech.inlineforms.movement.old; Kuka.IsGlobalPoint=False; Kuka.PointName=P366; Kuka.BlendingEnabled=TRUE; Kuka.MoveDataName=CPDATP366; Kuka.VelocityPath=1; Kuka.CurrentCDSetIndex=0; Kuka.MovementParameterFieldEnabled=True; IlfCommand=LIN
;ENDFOLD
$BWDSTART = FALSE
LDAT_ACT=LCPDATP366
FDAT_ACT=FP366
BAS (#CP_PARAMS,1)
SET_CD_PARAMS (0)
LIN XP366 C_DIS

;ENDFOLD
;FOLD LIN P367 CONT Vel=1 m/s CPDATP367 Tool[2] Base[10] ;%{PE}
;FOLD Parameters ;%{h}
;Params IlfProvider=kukaroboter.basistech.inlineforms.movement.old; Kuka.IsGlobalPoint=False; Kuka.PointName=P367; Kuka.BlendingEnabled=TRUE; Kuka.MoveDataName=CPDATP367; Kuka.VelocityPath=1; Kuka.CurrentCDSetIndex=0; Kuka.MovementParameterFieldEnabled=True; IlfCommand=LIN
;ENDFOLD
$BWDSTART = FALSE
LDAT_ACT=LCPDATP367
FDAT_ACT=FP367
BAS (#CP_PARAMS,1)
SET_CD_PARAMS (0)
LIN XP367 C_DIS

;ENDFOLD
;FOLD CIRC CAux368 CDes368 CONT Vel=0.1 m/s CPDATC368 Tool[2] Base[10] ;%{PE}
;FOLD Parameters ;%{h}
;Params IlfProvider=kukaroboter.basistech.inlineforms.movement.old; Kuka.IsGlobalPoint=False; Kuka.PointName=CDes368; Kuka.BlendingEnabled=TRUE; Kuka.MoveDataName=CPDATC368; Kuka.VelocityPath=0.1; Kuka.CurrentCDSetIndex=0; Kuka.MovementParameterFieldEnabled=True; IlfCommand=LIN
;ENDFOLD
$BWDSTART = FALSE
LDAT_ACT=LCPDATC368
FDAT_ACT=FC368
$ORI_TYPE = #VAR
$CIRC_TYPE = #PATH
BAS (#CP_PARAMS,0.1)
SET_CD_PARAMS (0)
CIRC XCAux368, XCDes368 C_DIS

;ENDFOLD
;FOLD LIN P369 CONT Vel=1 m/s CPDATP369 Tool[2] Base[10] ;%{PE}
;FOLD Parameters ;%{h}
;Params IlfProvider=kukaroboter.basistech.inlineforms.movement.old; Kuka.IsGlobalPoint=False; Kuka.PointName=P369; Kuka.BlendingEnabled=TRUE; Kuka.MoveDataName=CPDATP369; Kuka.VelocityPath=1; Kuka.CurrentCDSetIndex=0; Kuka.MovementParameterFieldEnabled=True; IlfCommand=LIN
;ENDFOLD
$BWDSTART = FALSE
LDAT_ACT=LCPDATP369
FDAT_ACT=FP369
BAS (#CP_PARAMS,1)
SET_CD_PARAMS (0)
LIN XP369 C_DIS

;ENDFOLD
;FOLD LIN P370 CONT Vel=1 m/s CPDATP370 Tool[2] Base[10] ;%{PE}
;FOLD Parameters ;%{h}
;Params IlfProvider=kukaroboter.basistech.inlineforms.movement.old; Kuka.IsGlobalPoint=False; Kuka.PointName=P370; Kuka.BlendingEnabled=TRUE; Kuka.MoveDataName=CPDATP370; Kuka.VelocityPath=1; Kuka.CurrentCDSetIndex=0; Kuka.MovementParameterFieldEnabled=True; IlfCommand=LIN
;ENDFOLD
$BWDSTART = FALSE
LDAT_ACT=LCPDATP370
FDAT_ACT=FP370
BAS (#CP_PARAMS,1)
SET_CD_PARAMS (0)
LIN XP370 C_DIS

;ENDFOLD
;FOLD CIRC CAux371 CDes371 CONT Vel=0.1 m/s CPDATC371 Tool[2] Base[10] ;%{PE}
;FOLD Parameters ;%{h}
;Params IlfProvider=kukaroboter.basistech.inlineforms.movement.old; Kuka.IsGlobalPoint=False; Kuka.PointName=CDes371; Kuka.BlendingEnabled=TRUE; Kuka.MoveDataName=CPDATC371; Kuka.VelocityPath=0.1; Kuka.CurrentCDSetIndex=0; Kuka.MovementParameterFieldEnabled=True; IlfCommand=LIN
;ENDFOLD
$BWDSTART = FALSE
LDAT_ACT=LCPDATC371
FDAT_ACT=FC371
$ORI_TYPE = #VAR
$CIRC_TYPE = #PATH
BAS (#CP_PARAMS,0.1)
SET_CD_PARAMS (0)
CIRC XCAux371, XCDes371 C_DIS

;ENDFOLD
;FOLD LIN P372 CONT Vel=1 m/s CPDATP372 Tool[2] Base[10] ;%{PE}
;FOLD Parameters ;%{h}
;Params IlfProvider=kukaroboter.basistech.inlineforms.movement.old; Kuka.IsGlobalPoint=False; Kuka.PointName=P372; Kuka.BlendingEnabled=TRUE; Kuka.MoveDataName=CPDATP372; Kuka.VelocityPath=1; Kuka.CurrentCDSetIndex=0; Kuka.MovementParameterFieldEnabled=True; IlfCommand=LIN
;ENDFOLD
$BWDSTART = FALSE
LDAT_ACT=LCPDATP372
FDAT_ACT=FP372
BAS (#CP_PARAMS,1)
SET_CD_PARAMS (0)
LIN XP372 C_DIS

;ENDFOLD
;FOLD LIN P373 CONT Vel=1 m/s CPDATP373 Tool[2] Base[10] ;%{PE}
;FOLD Parameters ;%{h}
;Params IlfProvider=kukaroboter.basistech.inlineforms.movement.old; Kuka.IsGlobalPoint=False; Kuka.PointName=P373; Kuka.BlendingEnabled=TRUE; Kuka.MoveDataName=CPDATP373; Kuka.VelocityPath=1; Kuka.CurrentCDSetIndex=0; Kuka.MovementParameterFieldEnabled=True; IlfCommand=LIN
;ENDFOLD
$BWDSTART = FALSE
LDAT_ACT=LCPDATP373
FDAT_ACT=FP373
BAS (#CP_PARAMS,1)
SET_CD_PARAMS (0)
LIN XP373 C_DIS

;ENDFOLD
;FOLD CIRC CAux374 CDes374 CONT Vel=0.1 m/s CPDATC374 Tool[2] Base[10] ;%{PE}
;FOLD Parameters ;%{h}
;Params IlfProvider=kukaroboter.basistech.inlineforms.movement.old; Kuka.IsGlobalPoint=False; Kuka.PointName=CDes374; Kuka.BlendingEnabled=TRUE; Kuka.MoveDataName=CPDATC374; Kuka.VelocityPath=0.1; Kuka.CurrentCDSetIndex=0; Kuka.MovementParameterFieldEnabled=True; IlfCommand=LIN
;ENDFOLD
$BWDSTART = FALSE
LDAT_ACT=LCPDATC374
FDAT_ACT=FC374
$ORI_TYPE = #VAR
$CIRC_TYPE = #PATH
BAS (#CP_PARAMS,0.1)
SET_CD_PARAMS (0)
CIRC XCAux374, XCDes374 C_DIS

;ENDFOLD
;FOLD LIN P375 CONT Vel=1 m/s CPDATP375 Tool[2] Base[10] ;%{PE}
;FOLD Parameters ;%{h}
;Params IlfProvider=kukaroboter.basistech.inlineforms.movement.old; Kuka.IsGlobalPoint=False; Kuka.PointName=P375; Kuka.BlendingEnabled=TRUE; Kuka.MoveDataName=CPDATP375; Kuka.VelocityPath=1; Kuka.CurrentCDSetIndex=0; Kuka.MovementParameterFieldEnabled=True; IlfCommand=LIN
;ENDFOLD
$BWDSTART = FALSE
LDAT_ACT=LCPDATP375
FDAT_ACT=FP375
BAS (#CP_PARAMS,1)
SET_CD_PARAMS (0)
LIN XP375 C_DIS

;ENDFOLD
;FOLD LIN P376 CONT Vel=1 m/s CPDATP376 Tool[2] Base[10] ;%{PE}
;FOLD Parameters ;%{h}
;Params IlfProvider=kukaroboter.basistech.inlineforms.movement.old; Kuka.IsGlobalPoint=False; Kuka.PointName=P376; Kuka.BlendingEnabled=TRUE; Kuka.MoveDataName=CPDATP376; Kuka.VelocityPath=1; Kuka.CurrentCDSetIndex=0; Kuka.MovementParameterFieldEnabled=True; IlfCommand=LIN
;ENDFOLD
$BWDSTART = FALSE
LDAT_ACT=LCPDATP376
FDAT_ACT=FP376
BAS (#CP_PARAMS,1)
SET_CD_PARAMS (0)
LIN XP376 C_DIS

;ENDFOLD
;FOLD CIRC CAux377 CDes377 CONT Vel=0.1 m/s CPDATC377 Tool[2] Base[10] ;%{PE}
;FOLD Parameters ;%{h}
;Params IlfProvider=kukaroboter.basistech.inlineforms.movement.old; Kuka.IsGlobalPoint=False; Kuka.PointName=CDes377; Kuka.BlendingEnabled=TRUE; Kuka.MoveDataName=CPDATC377; Kuka.VelocityPath=0.1; Kuka.CurrentCDSetIndex=0; Kuka.MovementParameterFieldEnabled=True; IlfCommand=LIN
;ENDFOLD
$BWDSTART = FALSE
LDAT_ACT=LCPDATC377
FDAT_ACT=FC377
$ORI_TYPE = #VAR
$CIRC_TYPE = #PATH
BAS (#CP_PARAMS,0.1)
SET_CD_PARAMS (0)
CIRC XCAux377, XCDes377 C_DIS

;ENDFOLD
;FOLD LIN P378 CONT Vel=1 m/s CPDATP378 Tool[2] Base[10] ;%{PE}
;FOLD Parameters ;%{h}
;Params IlfProvider=kukaroboter.basistech.inlineforms.movement.old; Kuka.IsGlobalPoint=False; Kuka.PointName=P378; Kuka.BlendingEnabled=TRUE; Kuka.MoveDataName=CPDATP378; Kuka.VelocityPath=1; Kuka.CurrentCDSetIndex=0; Kuka.MovementParameterFieldEnabled=True; IlfCommand=LIN
;ENDFOLD
$BWDSTART = FALSE
LDAT_ACT=LCPDATP378
FDAT_ACT=FP378
BAS (#CP_PARAMS,1)
SET_CD_PARAMS (0)
LIN XP378 C_DIS

;ENDFOLD
;FOLD LIN P379 CONT Vel=1 m/s CPDATP379 Tool[2] Base[10] ;%{PE}
;FOLD Parameters ;%{h}
;Params IlfProvider=kukaroboter.basistech.inlineforms.movement.old; Kuka.IsGlobalPoint=False; Kuka.PointName=P379; Kuka.BlendingEnabled=TRUE; Kuka.MoveDataName=CPDATP379; Kuka.VelocityPath=1; Kuka.CurrentCDSetIndex=0; Kuka.MovementParameterFieldEnabled=True; IlfCommand=LIN
;ENDFOLD
$BWDSTART = FALSE
LDAT_ACT=LCPDATP379
FDAT_ACT=FP379
BAS (#CP_PARAMS,1)
SET_CD_PARAMS (0)
LIN XP379 C_DIS

;ENDFOLD
;FOLD CIRC CAux380 CDes380 CONT Vel=0.1 m/s CPDATC380 Tool[2] Base[10] ;%{PE}
;FOLD Parameters ;%{h}
;Params IlfProvider=kukaroboter.basistech.inlineforms.movement.old; Kuka.IsGlobalPoint=False; Kuka.PointName=CDes380; Kuka.BlendingEnabled=TRUE; Kuka.MoveDataName=CPDATC380; Kuka.VelocityPath=0.1; Kuka.CurrentCDSetIndex=0; Kuka.MovementParameterFieldEnabled=True; IlfCommand=LIN
;ENDFOLD
$BWDSTART = FALSE
LDAT_ACT=LCPDATC380
FDAT_ACT=FC380
$ORI_TYPE = #VAR
$CIRC_TYPE = #PATH
BAS (#CP_PARAMS,0.1)
SET_CD_PARAMS (0)
CIRC XCAux380, XCDes380 C_DIS

;ENDFOLD
;FOLD LIN P381 CONT Vel=1 m/s CPDATP381 Tool[2] Base[10] ;%{PE}
;FOLD Parameters ;%{h}
;Params IlfProvider=kukaroboter.basistech.inlineforms.movement.old; Kuka.IsGlobalPoint=False; Kuka.PointName=P381; Kuka.BlendingEnabled=TRUE; Kuka.MoveDataName=CPDATP381; Kuka.VelocityPath=1; Kuka.CurrentCDSetIndex=0; Kuka.MovementParameterFieldEnabled=True; IlfCommand=LIN
;ENDFOLD
$BWDSTART = FALSE
LDAT_ACT=LCPDATP381
FDAT_ACT=FP381
BAS (#CP_PARAMS,1)
SET_CD_PARAMS (0)
LIN XP381 C_DIS

;ENDFOLD
;FOLD LIN P382 CONT Vel=1 m/s CPDATP382 Tool[2] Base[10] ;%{PE}
;FOLD Parameters ;%{h}
;Params IlfProvider=kukaroboter.basistech.inlineforms.movement.old; Kuka.IsGlobalPoint=False; Kuka.PointName=P382; Kuka.BlendingEnabled=TRUE; Kuka.MoveDataName=CPDATP382; Kuka.VelocityPath=1; Kuka.CurrentCDSetIndex=0; Kuka.MovementParameterFieldEnabled=True; IlfCommand=LIN
;ENDFOLD
$BWDSTART = FALSE
LDAT_ACT=LCPDATP382
FDAT_ACT=FP382
BAS (#CP_PARAMS,1)
SET_CD_PARAMS (0)
LIN XP382 C_DIS

;ENDFOLD
;FOLD CIRC CAux383 CDes383 CONT Vel=0.1 m/s CPDATC383 Tool[2] Base[10] ;%{PE}
;FOLD Parameters ;%{h}
;Params IlfProvider=kukaroboter.basistech.inlineforms.movement.old; Kuka.IsGlobalPoint=False; Kuka.PointName=CDes383; Kuka.BlendingEnabled=TRUE; Kuka.MoveDataName=CPDATC383; Kuka.VelocityPath=0.1; Kuka.CurrentCDSetIndex=0; Kuka.MovementParameterFieldEnabled=True; IlfCommand=LIN
;ENDFOLD
$BWDSTART = FALSE
LDAT_ACT=LCPDATC383
FDAT_ACT=FC383
$ORI_TYPE = #VAR
$CIRC_TYPE = #PATH
BAS (#CP_PARAMS,0.1)
SET_CD_PARAMS (0)
CIRC XCAux383, XCDes383 C_DIS

;ENDFOLD
;FOLD LIN P384 CONT Vel=1 m/s CPDATP384 Tool[2] Base[10] ;%{PE}
;FOLD Parameters ;%{h}
;Params IlfProvider=kukaroboter.basistech.inlineforms.movement.old; Kuka.IsGlobalPoint=False; Kuka.PointName=P384; Kuka.BlendingEnabled=TRUE; Kuka.MoveDataName=CPDATP384; Kuka.VelocityPath=1; Kuka.CurrentCDSetIndex=0; Kuka.MovementParameterFieldEnabled=True; IlfCommand=LIN
;ENDFOLD
$BWDSTART = FALSE
LDAT_ACT=LCPDATP384
FDAT_ACT=FP384
BAS (#CP_PARAMS,1)
SET_CD_PARAMS (0)
LIN XP384 C_DIS

;ENDFOLD
;FOLD LIN P385 CONT Vel=1 m/s CPDATP385 Tool[2] Base[10] ;%{PE}
;FOLD Parameters ;%{h}
;Params IlfProvider=kukaroboter.basistech.inlineforms.movement.old; Kuka.IsGlobalPoint=False; Kuka.PointName=P385; Kuka.BlendingEnabled=TRUE; Kuka.MoveDataName=CPDATP385; Kuka.VelocityPath=1; Kuka.CurrentCDSetIndex=0; Kuka.MovementParameterFieldEnabled=True; IlfCommand=LIN
;ENDFOLD
$BWDSTART = FALSE
LDAT_ACT=LCPDATP385
FDAT_ACT=FP385
BAS (#CP_PARAMS,1)
SET_CD_PARAMS (0)
LIN XP385 C_DIS

;ENDFOLD
;FOLD CIRC CAux386 CDes386 CONT Vel=0.1 m/s CPDATC386 Tool[2] Base[10] ;%{PE}
;FOLD Parameters ;%{h}
;Params IlfProvider=kukaroboter.basistech.inlineforms.movement.old; Kuka.IsGlobalPoint=False; Kuka.PointName=CDes386; Kuka.BlendingEnabled=TRUE; Kuka.MoveDataName=CPDATC386; Kuka.VelocityPath=0.1; Kuka.CurrentCDSetIndex=0; Kuka.MovementParameterFieldEnabled=True; IlfCommand=LIN
;ENDFOLD
$BWDSTART = FALSE
LDAT_ACT=LCPDATC386
FDAT_ACT=FC386
$ORI_TYPE = #VAR
$CIRC_TYPE = #PATH
BAS (#CP_PARAMS,0.1)
SET_CD_PARAMS (0)
CIRC XCAux386, XCDes386 C_DIS

;ENDFOLD
;FOLD LIN P387 CONT Vel=1 m/s CPDATP387 Tool[2] Base[10] ;%{PE}
;FOLD Parameters ;%{h}
;Params IlfProvider=kukaroboter.basistech.inlineforms.movement.old; Kuka.IsGlobalPoint=False; Kuka.PointName=P387; Kuka.BlendingEnabled=TRUE; Kuka.MoveDataName=CPDATP387; Kuka.VelocityPath=1; Kuka.CurrentCDSetIndex=0; Kuka.MovementParameterFieldEnabled=True; IlfCommand=LIN
;ENDFOLD
$BWDSTART = FALSE
LDAT_ACT=LCPDATP387
FDAT_ACT=FP387
BAS (#CP_PARAMS,1)
SET_CD_PARAMS (0)
LIN XP387 C_DIS

;ENDFOLD
;FOLD LIN P388 CONT Vel=1 m/s CPDATP388 Tool[2] Base[10] ;%{PE}
;FOLD Parameters ;%{h}
;Params IlfProvider=kukaroboter.basistech.inlineforms.movement.old; Kuka.IsGlobalPoint=False; Kuka.PointName=P388; Kuka.BlendingEnabled=TRUE; Kuka.MoveDataName=CPDATP388; Kuka.VelocityPath=1; Kuka.CurrentCDSetIndex=0; Kuka.MovementParameterFieldEnabled=True; IlfCommand=LIN
;ENDFOLD
$BWDSTART = FALSE
LDAT_ACT=LCPDATP388
FDAT_ACT=FP388
BAS (#CP_PARAMS,1)
SET_CD_PARAMS (0)
LIN XP388 C_DIS

